Yaskawa INFORM job: A_ROOF_UPPER_0614_2_PAINT_65.JBI

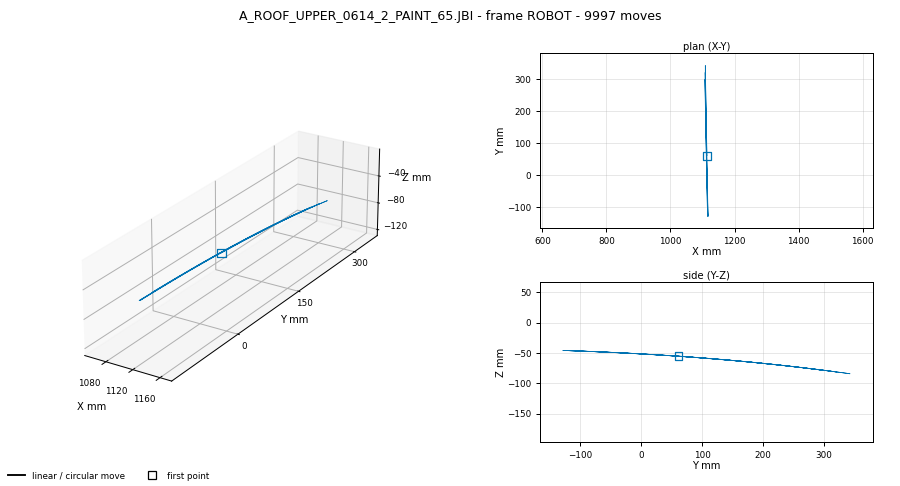
[picture p0: tool path of A_ROOF_UPPER_0614_2_PAINT_65.JBI in frame ROBOT, 9997 of 9997 moves have a stored position in this frame; points joined in program order, loops and branches not executed]
/JOB
//NAME A_ROOF_UPPER_0614_2_PAINT65
//POS
///NPOS 9997,0,0,0,0,0
///TOOL 1
///USER 0
///POSTYPE ROBOT
///RECTAN
///RCONF 1,0,0,0,0,0,0,0,0,0,0,0,0,0,0,0,0,0,0,0,0,0,0,0
C00000=1113.862,60.934,-55.122,179.977,7.455,149.407
C00001=1113.858,61.184,-55.139,179.979,7.459,149.407
C00002=1113.853,61.433,-55.156,179.980,7.462,149.408
C00003=1113.849,61.682,-55.174,179.981,7.466,149.408
C00004=1113.843,61.932,-55.191,179.983,7.470,149.409
C00005=1113.839,62.182,-55.208,179.984,7.475,149.409
C00006=1113.833,62.431,-55.225,179.985,7.478,149.410
C00007=1113.829,62.679,-55.242,179.986,7.483,149.410
C00008=1113.824,62.929,-55.259,179.988,7.487,149.411
C00009=1113.819,63.179,-55.276,179.989,7.491,149.411
C00010=1113.815,63.393,-55.291,179.990,7.494,149.412
C00011=1113.810,63.608,-55.306,179.991,7.497,149.412
C00012=1113.806,63.821,-55.321,179.992,7.500,149.413
C00013=1113.802,64.035,-55.336,179.993,7.504,149.413
C00014=1113.798,64.250,-55.351,179.994,7.507,149.414
C00015=1113.794,64.464,-55.366,179.995,7.510,149.414
C00016=1113.790,64.677,-55.380,179.997,7.514,149.415
C00017=1113.785,64.892,-55.395,179.998,7.518,149.415
C00018=1113.781,65.142,-55.412,179.999,7.521,149.415
C00019=1113.776,65.391,-55.429,-180.000,7.526,149.416
C00020=1113.771,65.641,-55.447,-179.998,7.530,149.417
C00021=1113.766,65.889,-55.464,-179.996,7.534,149.417
C00022=1113.761,66.138,-55.482,-179.995,7.538,149.418
C00023=1113.756,66.388,-55.499,-179.994,7.541,149.418
C00024=1113.751,66.637,-55.516,-179.993,7.545,149.418
C00025=1113.746,66.887,-55.533,-179.992,7.549,149.419
C00026=1113.741,67.136,-55.551,-179.990,7.553,149.420
C00027=1113.737,67.386,-55.568,-179.989,7.557,149.420
C00028=1113.732,67.635,-55.586,-179.987,7.561,149.421
C00029=1113.727,67.885,-55.603,-179.986,7.565,149.421
C00030=1113.722,68.134,-55.621,-179.985,7.569,149.422
C00031=1113.717,68.383,-55.638,-179.983,7.573,149.422
C00032=1113.712,68.632,-55.656,-179.982,7.576,149.423
C00033=1113.707,68.882,-55.673,-179.981,7.581,149.423
C00034=1113.702,69.131,-55.691,-179.980,7.585,149.424
C00035=1113.698,69.380,-55.709,-179.978,7.589,149.424
C00036=1113.693,69.630,-55.726,-179.976,7.592,149.425
C00037=1113.688,69.879,-55.744,-179.975,7.597,149.425
C00038=1113.682,70.128,-55.761,-179.974,7.601,149.426
C00039=1113.677,70.377,-55.779,-179.972,7.605,149.426
C00040=1113.673,70.626,-55.796,-179.971,7.609,149.427
C00041=1113.668,70.876,-55.813,-179.969,7.613,149.427
C00042=1113.663,71.125,-55.831,-179.969,7.616,149.428
C00043=1113.658,71.374,-55.849,-179.967,7.620,149.428
C00044=1113.653,71.625,-55.867,-179.966,7.624,149.429
C00045=1113.649,71.874,-55.884,-179.964,7.628,149.429
C00046=1113.644,72.123,-55.902,-179.963,7.632,149.430
C00047=1113.639,72.373,-55.920,-179.962,7.636,149.430
C00048=1113.634,72.622,-55.938,-179.960,7.640,149.431
C00049=1113.629,72.871,-55.956,-179.958,7.644,149.431
C00050=1113.624,73.120,-55.974,-179.957,7.648,149.432
C00051=1113.619,73.370,-55.991,-179.956,7.652,149.432
C00052=1113.614,73.619,-56.009,-179.954,7.656,149.433
C00053=1113.610,73.868,-56.026,-179.953,7.660,149.433
C00054=1113.605,74.117,-56.044,-179.952,7.663,149.434
C00055=1113.600,74.367,-56.062,-179.950,7.667,149.434
C00056=1113.595,74.616,-56.079,-179.949,7.671,149.434
C00057=1113.590,74.866,-56.097,-179.948,7.675,149.435
C00058=1113.585,75.115,-56.115,-179.946,7.679,149.436
C00059=1113.580,75.364,-56.133,-179.945,7.683,149.436
C00060=1113.575,75.613,-56.151,-179.944,7.688,149.437
C00061=1113.570,75.862,-56.169,-179.942,7.691,149.437
C00062=1113.566,76.113,-56.187,-179.940,7.695,149.437
C00063=1113.561,76.362,-56.205,-179.939,7.699,149.438
C00064=1113.556,76.611,-56.223,-179.938,7.704,149.439
C00065=1113.551,76.860,-56.241,-179.936,7.707,149.439
C00066=1113.547,77.074,-56.257,-179.935,7.711,149.439
C00067=1113.543,77.288,-56.272,-179.934,7.714,149.440
C00068=1113.539,77.503,-56.287,-179.934,7.717,149.441
C00069=1113.535,77.716,-56.303,-179.933,7.720,149.441
C00070=1113.531,77.931,-56.318,-179.932,7.723,149.441
C00071=1113.526,78.144,-56.334,-179.931,7.726,149.442
C00072=1113.522,78.359,-56.349,-179.930,7.729,149.442
C00073=1113.518,78.572,-56.365,-179.930,7.732,149.443
C00074=1113.513,78.822,-56.383,-179.928,7.736,149.443
C00075=1113.508,79.071,-56.401,-179.928,7.740,149.444
C00076=1113.504,79.321,-56.419,-179.926,7.744,149.444
C00077=1113.499,79.570,-56.437,-179.926,7.747,149.445
C00078=1113.494,79.819,-56.455,-179.924,7.751,149.445
C00079=1113.489,80.068,-56.473,-179.924,7.755,149.446
C00080=1113.484,80.317,-56.491,-179.922,7.758,149.447
C00081=1113.480,80.567,-56.509,-179.921,7.763,149.447
C00082=1113.475,80.816,-56.527,-179.920,7.766,149.448
C00083=1113.469,81.066,-56.546,-179.919,7.770,149.448
C00084=1113.464,81.315,-56.564,-179.918,7.773,149.449
C00085=1113.459,81.564,-56.582,-179.917,7.777,149.449
C00086=1113.455,81.814,-56.600,-179.916,7.781,149.450
C00087=1113.450,82.063,-56.618,-179.915,7.785,149.450
C00088=1113.445,82.312,-56.636,-179.914,7.788,149.451
C00089=1113.440,82.561,-56.655,-179.913,7.792,149.452
C00090=1113.436,82.810,-56.673,-179.911,7.796,149.452
C00091=1113.430,83.060,-56.692,-179.911,7.800,149.453
C00092=1113.426,83.310,-56.710,-179.909,7.804,149.453
C00093=1113.421,83.559,-56.728,-179.908,7.807,149.454
C00094=1113.416,83.808,-56.746,-179.907,7.811,149.454
C00095=1113.412,84.057,-56.765,-179.906,7.815,149.455
C00096=1113.407,84.306,-56.783,-179.905,7.818,149.455
C00097=1113.401,84.556,-56.801,-179.904,7.823,149.456
C00098=1113.396,84.805,-56.819,-179.902,7.827,149.456
C00099=1113.392,85.055,-56.838,-179.901,7.830,149.457
C00100=1113.387,85.303,-56.856,-179.900,7.834,149.457
C00101=1113.382,85.553,-56.874,-179.898,7.838,149.458
C00102=1113.377,85.802,-56.893,-179.898,7.841,149.458
C00103=1113.372,86.052,-56.911,-179.896,7.845,149.459
C00104=1113.368,86.301,-56.930,-179.895,7.849,149.459
C00105=1113.363,86.550,-56.948,-179.894,7.853,149.460
C00106=1113.357,86.799,-56.967,-179.893,7.856,149.460
C00107=1113.353,87.048,-56.986,-179.891,7.860,149.461
C00108=1113.348,87.298,-57.004,-179.890,7.864,149.461
C00109=1113.343,87.547,-57.022,-179.889,7.868,149.462
C00110=1113.339,87.796,-57.041,-179.887,7.872,149.462
C00111=1113.334,88.046,-57.059,-179.886,7.876,149.463
C00112=1113.329,88.295,-57.077,-179.885,7.879,149.463
C00113=1113.324,88.544,-57.097,-179.884,7.883,149.464
C00114=1113.319,88.793,-57.115,-179.882,7.887,149.464
C00115=1113.314,89.043,-57.133,-179.881,7.891,149.465
C00116=1113.310,89.292,-57.152,-179.880,7.894,149.465
C00117=1113.305,89.541,-57.170,-179.879,7.898,149.466
C00118=1113.300,89.790,-57.189,-179.877,7.902,149.466
C00119=1113.295,90.040,-57.208,-179.876,7.906,149.467
C00120=1113.290,90.289,-57.226,-179.875,7.909,149.467
C00121=1113.286,90.538,-57.245,-179.873,7.914,149.468
C00122=1113.282,90.752,-57.261,-179.872,7.916,149.468
C00123=1113.277,90.966,-57.277,-179.870,7.920,149.469
C00124=1113.273,91.180,-57.294,-179.869,7.923,149.469
C00125=1113.269,91.394,-57.309,-179.868,7.926,149.469
C00126=1113.265,91.609,-57.325,-179.867,7.930,149.470
C00127=1113.261,91.823,-57.341,-179.866,7.933,149.470
C00128=1113.257,92.036,-57.357,-179.865,7.937,149.471
C00129=1113.252,92.250,-57.373,-179.864,7.940,149.471
C00130=1113.248,92.500,-57.392,-179.862,7.944,149.472
C00131=1113.242,92.749,-57.411,-179.861,7.947,149.472
C00132=1113.238,92.998,-57.430,-179.859,7.951,149.472
C00133=1113.234,93.247,-57.449,-179.858,7.955,149.473
C00134=1113.228,93.497,-57.467,-179.856,7.959,149.473
C00135=1113.224,93.746,-57.486,-179.855,7.962,149.474
C00136=1113.218,93.995,-57.505,-179.854,7.967,149.474
C00137=1113.214,94.244,-57.524,-179.852,7.970,149.475
C00138=1113.209,94.493,-57.543,-179.851,7.974,149.475
C00139=1113.204,94.743,-57.561,-179.849,7.978,149.476
C00140=1113.199,94.992,-57.581,-179.847,7.982,149.476
C00141=1113.194,95.241,-57.599,-179.846,7.986,149.477
C00142=1113.190,95.491,-57.618,-179.844,7.990,149.477
C00143=1113.185,95.739,-57.637,-179.843,7.993,149.477
C00144=1113.180,95.989,-57.657,-179.842,7.997,149.478
C00145=1113.175,96.238,-57.675,-179.840,8.001,149.478
C00146=1113.171,96.488,-57.694,-179.838,8.005,149.479
C00147=1113.166,96.736,-57.713,-179.837,8.009,149.479
C00148=1113.160,96.986,-57.732,-179.835,8.012,149.480
C00149=1113.156,97.235,-57.751,-179.834,8.016,149.480
C00150=1113.151,97.484,-57.770,-179.832,8.020,149.481
C00151=1113.146,97.733,-57.790,-179.830,8.024,149.481
C00152=1113.141,97.983,-57.808,-179.829,8.028,149.481
C00153=1113.137,98.232,-57.827,-179.827,8.032,149.482
C00154=1113.132,98.481,-57.846,-179.825,8.035,149.482
C00155=1113.127,98.730,-57.866,-179.824,8.039,149.482
C00156=1113.123,98.980,-57.885,-179.822,8.043,149.483
C00157=1113.118,99.229,-57.903,-179.821,8.046,149.483
C00158=1113.113,99.479,-57.923,-179.819,8.050,149.484
C00159=1113.108,99.727,-57.942,-179.818,8.054,149.484
C00160=1113.104,99.977,-57.961,-179.816,8.058,149.485
C00161=1113.098,100.226,-57.981,-179.814,8.061,149.485
C00162=1113.094,100.475,-58.000,-179.813,8.065,149.485
C00163=1113.089,100.724,-58.019,-179.811,8.069,149.486
C00164=1113.084,100.973,-58.039,-179.809,8.073,149.486
C00165=1113.080,101.222,-58.057,-179.807,8.077,149.486
C00166=1113.075,101.471,-58.077,-179.806,8.080,149.487
C00167=1113.070,101.722,-58.096,-179.804,8.084,149.487
C00168=1113.065,101.970,-58.115,-179.802,8.088,149.488
C00169=1113.060,102.220,-58.134,-179.800,8.092,149.488
C00170=1113.055,102.469,-58.154,-179.799,8.096,149.488
C00171=1113.050,102.718,-58.173,-179.797,8.099,149.489
C00172=1113.046,102.967,-58.192,-179.795,8.103,149.489
C00173=1113.041,103.216,-58.212,-179.794,8.107,149.489
C00174=1113.036,103.466,-58.231,-179.792,8.111,149.490
C00175=1113.031,103.715,-58.251,-179.790,8.114,149.490
C00176=1113.027,103.963,-58.270,-179.788,8.119,149.491
C00177=1113.022,104.213,-58.290,-179.786,8.122,149.491
C00178=1113.018,104.427,-58.307,-179.785,8.126,149.491
C00179=1113.014,104.640,-58.323,-179.783,8.129,149.491
C00180=1113.009,104.855,-58.340,-179.781,8.132,149.492
C00181=1113.005,105.069,-58.356,-179.780,8.135,149.492
C00182=1113.001,105.282,-58.373,-179.778,8.138,149.492
C00183=1112.997,105.497,-58.389,-179.777,8.141,149.492
C00184=1112.993,105.710,-58.407,-179.775,8.145,149.493
C00185=1112.989,105.924,-58.423,-179.774,8.148,149.493
C00186=1112.985,106.173,-58.443,-179.771,8.152,149.493
C00187=1112.980,106.422,-58.463,-179.769,8.156,149.494
C00188=1112.975,106.672,-58.482,-179.767,8.159,149.494
C00189=1112.970,106.921,-58.502,-179.766,8.163,149.494
C00190=1112.965,107.171,-58.522,-179.764,8.167,149.495
C00191=1112.960,107.419,-58.542,-179.762,8.170,149.495
C00192=1112.956,107.668,-58.561,-179.760,8.174,149.495
C00193=1112.952,107.918,-58.580,-179.758,8.178,149.496
C00194=1112.946,108.167,-58.600,-179.756,8.181,149.496
C00195=1112.942,108.416,-58.620,-179.754,8.185,149.496
C00196=1112.937,108.665,-58.640,-179.752,8.189,149.496
C00197=1112.932,108.915,-58.659,-179.750,8.193,149.497
C00198=1112.927,109.163,-58.679,-179.748,8.197,149.497
C00199=1112.922,109.413,-58.699,-179.746,8.200,149.497
C00200=1112.918,109.662,-58.719,-179.744,8.204,149.498
C00201=1112.913,109.911,-58.739,-179.742,8.207,149.498
C00202=1112.908,110.160,-58.758,-179.740,8.211,149.498
C00203=1112.903,110.410,-58.778,-179.738,8.215,149.498
C00204=1112.899,110.659,-58.798,-179.736,8.218,149.499
C00205=1112.894,110.908,-58.818,-179.733,8.222,149.499
C00206=1112.889,111.157,-58.837,-179.731,8.226,149.499
C00207=1112.884,111.406,-58.858,-179.730,8.229,149.500
C00208=1112.879,111.656,-58.877,-179.728,8.232,149.500
C00209=1112.875,111.905,-58.898,-179.726,8.236,149.500
C00210=1112.870,112.153,-58.917,-179.725,8.240,149.500
C00211=1112.865,112.402,-58.937,-179.723,8.243,149.501
C00212=1112.861,112.652,-58.957,-179.721,8.246,149.501
C00213=1112.856,112.901,-58.977,-179.719,8.250,149.501
C00214=1112.851,113.150,-58.997,-179.717,8.253,149.502
C00215=1112.847,113.399,-59.017,-179.715,8.257,149.502
C00216=1112.842,113.648,-59.037,-179.714,8.260,149.502
C00217=1112.837,113.897,-59.057,-179.712,8.264,149.502
C00218=1112.832,114.147,-59.077,-179.710,8.267,149.503
C00219=1112.827,114.396,-59.098,-179.709,8.271,149.503
C00220=1112.822,114.646,-59.117,-179.707,8.274,149.503
C00221=1112.818,114.895,-59.138,-179.705,8.277,149.504
C00222=1112.813,115.143,-59.157,-179.703,8.281,149.504
C00223=1112.808,115.392,-59.177,-179.701,8.285,149.504
C00224=1112.804,115.641,-59.198,-179.700,8.287,149.504
C00225=1112.798,115.891,-59.218,-179.698,8.291,149.505
C00226=1112.794,116.140,-59.238,-179.696,8.295,149.505
C00227=1112.789,116.389,-59.259,-179.694,8.298,149.505
C00228=1112.785,116.639,-59.278,-179.693,8.301,149.506
C00229=1112.780,116.888,-59.299,-179.691,8.304,149.506
C00230=1112.775,117.136,-59.319,-179.689,8.308,149.506
C00231=1112.770,117.386,-59.339,-179.687,8.312,149.506
C00232=1112.765,117.635,-59.359,-179.686,8.314,149.507
C00233=1112.761,117.884,-59.380,-179.684,8.318,149.507
C00234=1112.757,118.097,-59.397,-179.683,8.321,149.507
C00235=1112.752,118.311,-59.415,-179.681,8.324,149.508
C00236=1112.749,118.526,-59.432,-179.679,8.327,149.508
C00237=1112.745,118.739,-59.449,-179.678,8.330,149.508
C00238=1112.741,118.953,-59.467,-179.676,8.333,149.508
C00239=1112.737,119.167,-59.484,-179.675,8.335,149.508
C00240=1112.732,119.381,-59.501,-179.673,8.338,149.509
C00241=1112.728,119.594,-59.519,-179.671,8.342,149.509
C00242=1112.724,119.843,-59.539,-179.670,8.344,149.509
C00243=1112.719,120.093,-59.560,-179.668,8.348,149.510
C00244=1112.714,120.342,-59.580,-179.666,8.352,149.510
C00245=1112.709,120.591,-59.600,-179.665,8.354,149.510
C00246=1112.705,120.840,-59.621,-179.663,8.358,149.510
C00247=1112.700,121.089,-59.641,-179.661,8.362,149.511
C00248=1112.695,121.338,-59.662,-179.659,8.365,149.511
C00249=1112.691,121.587,-59.682,-179.658,8.368,149.511
C00250=1112.686,121.836,-59.703,-179.655,8.372,149.511
C00251=1112.681,122.085,-59.724,-179.654,8.375,149.512
C00252=1112.677,122.335,-59.743,-179.652,8.378,149.512
C00253=1112.671,122.584,-59.764,-179.650,8.382,149.512
C00254=1112.667,122.833,-59.785,-179.648,8.385,149.513
C00255=1112.663,123.082,-59.805,-179.647,8.388,149.513
C00256=1112.657,123.331,-59.826,-179.645,8.392,149.513
C00257=1112.653,123.580,-59.846,-179.643,8.395,149.513
C00258=1112.648,123.830,-59.867,-179.641,8.399,149.514
C00259=1112.643,124.079,-59.888,-179.640,8.402,149.514
C00260=1112.639,124.328,-59.908,-179.638,8.405,149.514
C00261=1112.634,124.577,-59.929,-179.636,8.409,149.515
C00262=1112.629,124.826,-59.949,-179.635,8.412,149.515
C00263=1112.624,125.075,-59.970,-179.633,8.415,149.515
C00264=1112.620,125.324,-59.991,-179.631,8.419,149.515
C00265=1112.615,125.573,-60.011,-179.629,8.422,149.516
C00266=1112.611,125.823,-60.032,-179.627,8.425,149.516
C00267=1112.606,126.072,-60.053,-179.626,8.429,149.516
C00268=1112.601,126.320,-60.074,-179.624,8.432,149.517
C00269=1112.597,126.569,-60.095,-179.622,8.435,149.517
C00270=1112.592,126.819,-60.116,-179.620,8.439,149.517
C00271=1112.587,127.068,-60.136,-179.619,8.441,149.517
C00272=1112.582,127.317,-60.157,-179.617,8.445,149.518
C00273=1112.578,127.566,-60.177,-179.615,8.449,149.518
C00274=1112.572,127.815,-60.198,-179.614,8.451,149.518
C00275=1112.568,128.064,-60.219,-179.611,8.455,149.518
C00276=1112.563,128.313,-60.240,-179.610,8.459,149.519
C00277=1112.559,128.562,-60.261,-179.608,8.462,149.519
C00278=1112.554,128.812,-60.282,-179.606,8.465,149.519
C00279=1112.550,129.060,-60.303,-179.604,8.469,149.519
C00280=1112.545,129.310,-60.324,-179.603,8.472,149.520
C00281=1112.540,129.558,-60.345,-179.601,8.475,149.520
C00282=1112.535,129.807,-60.366,-179.599,8.479,149.520
C00283=1112.530,130.057,-60.387,-179.597,8.482,149.521
C00284=1112.526,130.306,-60.407,-179.596,8.485,149.521
C00285=1112.521,130.555,-60.429,-179.594,8.489,149.521
C00286=1112.517,130.804,-60.449,-179.592,8.492,149.521
C00287=1112.512,131.053,-60.470,-179.591,8.495,149.522
C00288=1112.507,131.302,-60.491,-179.589,8.499,149.522
C00289=1112.502,131.551,-60.512,-179.587,8.502,149.522
C00290=1112.498,131.765,-60.531,-179.585,8.505,149.523
C00291=1112.494,131.979,-60.549,-179.584,8.508,149.523
C00292=1112.490,132.192,-60.567,-179.582,8.510,149.523
C00293=1112.487,132.406,-60.585,-179.581,8.513,149.523
C00294=1112.483,132.619,-60.603,-179.580,8.516,149.524
C00295=1112.478,132.834,-60.621,-179.579,8.519,149.524
C00296=1112.474,133.047,-60.639,-179.576,8.522,149.524
C00297=1112.470,133.261,-60.658,-179.575,8.525,149.524
C00298=1112.465,133.510,-60.678,-179.574,8.528,149.525
C00299=1112.461,133.759,-60.699,-179.572,8.531,149.525
C00300=1112.456,134.008,-60.721,-179.570,8.535,149.525
C00301=1112.451,134.257,-60.742,-179.568,8.538,149.526
C00302=1112.446,134.506,-60.764,-179.566,8.541,149.526
C00303=1112.442,134.755,-60.784,-179.565,8.545,149.526
C00304=1112.438,135.004,-60.806,-179.563,8.548,149.526
C00305=1112.432,135.254,-60.827,-179.561,8.552,149.527
C00306=1112.428,135.502,-60.848,-179.560,8.555,149.527
C00307=1112.423,135.751,-60.869,-179.558,8.558,149.527
C00308=1112.419,136.001,-60.891,-179.556,8.562,149.528
C00309=1112.414,136.250,-60.912,-179.554,8.565,149.528
C00310=1112.410,136.498,-60.933,-179.553,8.568,149.528
C00311=1112.404,136.747,-60.954,-179.551,8.572,149.528
C00312=1112.400,136.997,-60.976,-179.549,8.576,149.529
C00313=1112.395,137.246,-60.997,-179.548,8.578,149.529
C00314=1112.390,137.495,-61.019,-179.546,8.582,149.529
C00315=1112.386,137.744,-61.039,-179.544,8.586,149.530
C00316=1112.381,137.993,-61.061,-179.543,8.588,149.530
C00317=1112.377,138.242,-61.083,-179.541,8.592,149.530
C00318=1112.371,138.491,-61.104,-179.539,8.596,149.531
C00319=1112.367,138.740,-61.126,-179.538,8.598,149.531
C00320=1112.363,138.988,-61.147,-179.535,8.602,149.531
C00321=1112.358,139.238,-61.168,-179.534,8.606,149.532
C00322=1112.354,139.487,-61.190,-179.532,8.609,149.532
C00323=1112.349,139.736,-61.212,-179.531,8.612,149.532
C00324=1112.343,139.985,-61.233,-179.529,8.616,149.532
C00325=1112.339,140.234,-61.255,-179.527,8.619,149.533
C00326=1112.334,140.483,-61.276,-179.526,8.622,149.533
C00327=1112.330,140.732,-61.297,-179.524,8.626,149.533
C00328=1112.326,140.981,-61.319,-179.523,8.629,149.534
C00329=1112.321,141.230,-61.340,-179.520,8.633,149.534
C00330=1112.317,141.479,-61.363,-179.519,8.636,149.535
C00331=1112.311,141.729,-61.383,-179.517,8.639,149.535
C00332=1112.306,141.977,-61.405,-179.515,8.643,149.535
C00333=1112.302,142.226,-61.427,-179.514,8.646,149.535
C00334=1112.297,142.475,-61.449,-179.512,8.649,149.536
C00335=1112.292,142.724,-61.470,-179.511,8.653,149.536
C00336=1112.288,142.974,-61.492,-179.508,8.657,149.536
C00337=1112.283,143.222,-61.514,-179.507,8.660,149.537
C00338=1112.279,143.472,-61.536,-179.505,8.663,149.537
C00339=1112.274,143.720,-61.557,-179.504,8.667,149.537
C00340=1112.269,143.969,-61.579,-179.502,8.670,149.538
C00341=1112.265,144.218,-61.601,-179.501,8.674,149.538
C00342=1112.260,144.468,-61.622,-179.499,8.677,149.538
C00343=1112.255,144.717,-61.644,-179.497,8.681,149.539
C00344=1112.250,144.966,-61.666,-179.495,8.684,149.539
C00345=1112.246,145.215,-61.688,-179.494,8.687,149.539
C00346=1112.242,145.428,-61.706,-179.492,8.690,149.540
C00347=1112.238,145.642,-61.725,-179.490,8.694,149.540
C00348=1112.235,145.855,-61.744,-179.488,8.697,149.540
C00349=1112.230,146.069,-61.763,-179.487,8.700,149.540
C00350=1112.226,146.282,-61.781,-179.485,8.703,149.541
C00351=1112.222,146.496,-61.800,-179.483,8.706,149.541
C00352=1112.218,146.709,-61.818,-179.481,8.710,149.541
C00353=1112.214,146.924,-61.837,-179.480,8.712,149.541
C00354=1112.209,147.172,-61.859,-179.478,8.716,149.542
C00355=1112.205,147.422,-61.881,-179.476,8.719,149.542
C00356=1112.200,147.670,-61.903,-179.474,8.723,149.542
C00357=1112.196,147.920,-61.925,-179.471,8.727,149.542
C00358=1112.190,148.169,-61.947,-179.469,8.731,149.542
C00359=1112.187,148.417,-61.970,-179.467,8.734,149.543
C00360=1112.182,148.666,-61.992,-179.465,8.737,149.543
C00361=1112.177,148.915,-62.014,-179.462,8.741,149.543
C00362=1112.173,149.164,-62.035,-179.460,8.744,149.543
C00363=1112.168,149.413,-62.057,-179.458,8.748,149.544
C00364=1112.163,149.662,-62.079,-179.456,8.751,149.544
C00365=1112.158,149.912,-62.102,-179.454,8.755,149.544
C00366=1112.154,150.160,-62.123,-179.452,8.758,149.544
C00367=1112.150,150.409,-62.146,-179.450,8.762,149.545
C00368=1112.145,150.658,-62.168,-179.448,8.765,149.545
C00369=1112.140,150.907,-62.190,-179.446,8.769,149.545
C00370=1112.135,151.156,-62.212,-179.444,8.772,149.545
C00371=1112.131,151.405,-62.234,-179.442,8.776,149.546
C00372=1112.127,151.654,-62.257,-179.440,8.779,149.546
C00373=1112.122,151.903,-62.279,-179.438,8.783,149.546
C00374=1112.117,152.152,-62.301,-179.435,8.786,149.546
C00375=1112.112,152.401,-62.323,-179.433,8.789,149.546
C00376=1112.108,152.650,-62.346,-179.431,8.793,149.547
C00377=1112.103,152.899,-62.368,-179.429,8.796,149.547
C00378=1112.098,153.148,-62.390,-179.427,8.800,149.547
C00379=1112.094,153.397,-62.413,-179.425,8.803,149.547
C00380=1112.089,153.645,-62.434,-179.422,8.806,149.547
C00381=1112.084,153.895,-62.457,-179.420,8.810,149.548
C00382=1112.080,154.144,-62.480,-179.418,8.813,149.548
C00383=1112.075,154.392,-62.502,-179.416,8.817,149.548
C00384=1112.070,154.642,-62.524,-179.414,8.820,149.548
C00385=1112.066,154.890,-62.547,-179.412,8.823,149.548
C00386=1112.061,155.139,-62.569,-179.410,8.826,149.549
C00387=1112.057,155.388,-62.592,-179.408,8.830,149.549
C00388=1112.052,155.637,-62.614,-179.405,8.833,149.549
C00389=1112.047,155.887,-62.636,-179.403,8.836,149.549
C00390=1112.043,156.135,-62.659,-179.401,8.840,149.549
C00391=1112.038,156.384,-62.681,-179.398,8.843,149.549
C00392=1112.033,156.633,-62.704,-179.396,8.846,149.550
C00393=1112.029,156.882,-62.726,-179.394,8.850,149.550
C00394=1112.024,157.131,-62.749,-179.392,8.852,149.550
C00395=1112.020,157.380,-62.771,-179.390,8.856,149.550
C00396=1112.016,157.629,-62.794,-179.388,8.859,149.550
C00397=1112.011,157.878,-62.817,-179.386,8.862,149.550
C00398=1112.006,158.126,-62.839,-179.384,8.866,149.551
C00399=1112.001,158.376,-62.862,-179.382,8.869,149.551
C00400=1111.997,158.625,-62.884,-179.379,8.872,149.551
C00401=1111.992,158.873,-62.907,-179.378,8.875,149.551
C00402=1111.988,159.087,-62.927,-179.375,8.878,149.551
C00403=1111.985,159.301,-62.946,-179.374,8.881,149.551
C00404=1111.981,159.514,-62.966,-179.372,8.883,149.551
C00405=1111.976,159.727,-62.985,-179.370,8.887,149.552
C00406=1111.972,159.941,-63.004,-179.368,8.889,149.552
C00407=1111.969,160.155,-63.024,-179.366,8.892,149.552
C00408=1111.965,160.368,-63.044,-179.364,8.894,149.552
C00409=1111.960,160.581,-63.063,-179.362,8.898,149.552
C00410=1111.956,160.830,-63.085,-179.360,8.901,149.552
C00411=1111.951,161.079,-63.108,-179.358,8.903,149.552
C00412=1111.947,161.328,-63.132,-179.356,8.907,149.552
C00413=1111.942,161.577,-63.154,-179.354,8.910,149.553
C00414=1111.937,161.826,-63.177,-179.351,8.913,149.553
C00415=1111.933,162.075,-63.200,-179.349,8.917,149.553
C00416=1111.929,162.324,-63.223,-179.347,8.919,149.553
C00417=1111.924,162.573,-63.245,-179.345,8.922,149.553
C00418=1111.919,162.822,-63.268,-179.343,8.926,149.553
C00419=1111.914,163.071,-63.291,-179.341,8.929,149.553
C00420=1111.910,163.319,-63.314,-179.338,8.932,149.554
C00421=1111.906,163.568,-63.338,-179.336,8.934,149.554
C00422=1111.901,163.818,-63.360,-179.334,8.938,149.554
C00423=1111.897,164.067,-63.383,-179.332,8.941,149.554
C00424=1111.891,164.315,-63.406,-179.329,8.945,149.554
C00425=1111.887,164.564,-63.429,-179.328,8.947,149.554
C00426=1111.883,164.813,-63.452,-179.325,8.950,149.554
C00427=1111.878,165.062,-63.475,-179.323,8.953,149.554
C00428=1111.874,165.311,-63.498,-179.320,8.957,149.554
C00429=1111.869,165.560,-63.522,-179.319,8.959,149.555
C00430=1111.864,165.808,-63.545,-179.316,8.962,149.555
C00431=1111.860,166.057,-63.567,-179.314,8.966,149.555
C00432=1111.855,166.306,-63.590,-179.312,8.969,149.555
C00433=1111.850,166.555,-63.613,-179.310,8.971,149.555
C00434=1111.846,166.804,-63.637,-179.308,8.975,149.555
C00435=1111.842,167.053,-63.659,-179.305,8.978,149.555
C00436=1111.837,167.302,-63.683,-179.303,8.981,149.555
C00437=1111.832,167.551,-63.706,-179.301,8.984,149.556
C00438=1111.828,167.800,-63.729,-179.299,8.987,149.556
C00439=1111.823,168.048,-63.752,-179.297,8.990,149.556
C00440=1111.818,168.297,-63.775,-179.295,8.993,149.556
C00441=1111.814,168.546,-63.799,-179.292,8.996,149.556
C00442=1111.809,168.795,-63.822,-179.290,8.999,149.556
C00443=1111.805,169.044,-63.846,-179.288,9.002,149.556
C00444=1111.801,169.292,-63.869,-179.286,9.005,149.556
C00445=1111.796,169.541,-63.892,-179.284,9.008,149.556
C00446=1111.791,169.791,-63.916,-179.281,9.011,149.556
C00447=1111.786,170.040,-63.939,-179.280,9.014,149.557
C00448=1111.782,170.289,-63.962,-179.277,9.017,149.557
C00449=1111.778,170.537,-63.985,-179.275,9.020,149.557
C00450=1111.773,170.786,-64.008,-179.273,9.023,149.557
C00451=1111.769,171.035,-64.032,-179.271,9.026,149.557
C00452=1111.764,171.284,-64.056,-179.268,9.029,149.557
C00453=1111.759,171.533,-64.079,-179.266,9.033,149.557
C00454=1111.755,171.782,-64.103,-179.264,9.035,149.557
C00455=1111.750,172.031,-64.126,-179.262,9.038,149.557
C00456=1111.746,172.279,-64.150,-179.260,9.042,149.558
C00457=1111.741,172.528,-64.173,-179.258,9.044,149.558
C00458=1111.737,172.742,-64.193,-179.256,9.046,149.558
C00459=1111.733,172.955,-64.213,-179.253,9.049,149.558
C00460=1111.729,173.168,-64.233,-179.252,9.052,149.558
C00461=1111.725,173.382,-64.253,-179.250,9.054,149.558
C00462=1111.721,173.595,-64.273,-179.248,9.057,149.558
C00463=1111.717,173.808,-64.294,-179.247,9.059,149.558
C00464=1111.714,174.022,-64.314,-179.245,9.062,149.558
C00465=1111.709,174.235,-64.334,-179.243,9.064,149.558
C00466=1111.705,174.484,-64.358,-179.240,9.067,149.558
C00467=1111.700,174.733,-64.381,-179.238,9.071,149.559
C00468=1111.695,174.982,-64.405,-179.236,9.073,149.559
C00469=1111.691,175.230,-64.429,-179.234,9.076,149.559
C00470=1111.686,175.479,-64.452,-179.232,9.080,149.559
C00471=1111.682,175.728,-64.476,-179.230,9.082,149.559
C00472=1111.677,175.977,-64.500,-179.227,9.085,149.559
C00473=1111.673,176.227,-64.523,-179.225,9.089,149.559
C00474=1111.669,176.475,-64.547,-179.223,9.091,149.559
C00475=1111.664,176.724,-64.571,-179.221,9.094,149.559
C00476=1111.660,176.972,-64.595,-179.219,9.097,149.560
C00477=1111.655,177.221,-64.618,-179.217,9.100,149.560
C00478=1111.651,177.470,-64.642,-179.214,9.103,149.560
C00479=1111.646,177.719,-64.666,-179.212,9.106,149.560
C00480=1111.641,177.967,-64.690,-179.210,9.109,149.560
C00481=1111.637,178.216,-64.713,-179.208,9.112,149.560
C00482=1111.632,178.465,-64.737,-179.206,9.115,149.560
C00483=1111.628,178.714,-64.761,-179.204,9.118,149.560
C00484=1111.624,178.963,-64.785,-179.201,9.121,149.560
C00485=1111.619,179.212,-64.808,-179.200,9.123,149.561
C00486=1111.615,179.460,-64.832,-179.197,9.127,149.561
C00487=1111.609,179.710,-64.856,-179.195,9.130,149.561
C00488=1111.605,179.958,-64.880,-179.192,9.133,149.561
C00489=1111.601,180.207,-64.905,-179.190,9.136,149.561
C00490=1111.596,180.456,-64.928,-179.187,9.139,149.561
C00491=1111.592,180.705,-64.952,-179.185,9.142,149.561
C00492=1111.588,180.953,-64.976,-179.182,9.145,149.561
C00493=1111.583,181.202,-65.000,-179.180,9.148,149.561
C00494=1111.578,181.451,-65.024,-179.178,9.151,149.561
C00495=1111.574,181.700,-65.049,-179.176,9.154,149.561
C00496=1111.569,181.949,-65.072,-179.173,9.157,149.561
C00497=1111.565,182.197,-65.096,-179.171,9.160,149.561
C00498=1111.561,182.446,-65.120,-179.168,9.163,149.561
C00499=1111.555,182.695,-65.144,-179.166,9.167,149.561
C00500=1111.551,182.944,-65.169,-179.164,9.169,149.561
C00501=1111.547,183.193,-65.193,-179.161,9.172,149.561
C00502=1111.542,183.441,-65.217,-179.159,9.175,149.562
C00503=1111.537,183.690,-65.241,-179.156,9.178,149.562
C00504=1111.533,183.939,-65.265,-179.154,9.181,149.562
C00505=1111.529,184.188,-65.289,-179.152,9.184,149.562
C00506=1111.524,184.436,-65.313,-179.149,9.187,149.562
C00507=1111.519,184.685,-65.338,-179.147,9.190,149.562
C00508=1111.515,184.934,-65.361,-179.144,9.192,149.562
C00509=1111.511,185.183,-65.386,-179.142,9.195,149.562
C00510=1111.506,185.432,-65.411,-179.139,9.198,149.562
C00511=1111.501,185.680,-65.435,-179.137,9.200,149.562
C00512=1111.497,185.929,-65.459,-179.135,9.204,149.562
C00513=1111.492,186.178,-65.484,-179.132,9.207,149.562
C00514=1111.489,186.391,-65.504,-179.130,9.209,149.562
C00515=1111.485,186.604,-65.525,-179.129,9.211,149.562
C00516=1111.481,186.818,-65.547,-179.127,9.214,149.562
C00517=1111.477,187.031,-65.566,-179.125,9.216,149.562
C00518=1111.473,187.244,-65.587,-179.122,9.219,149.562
C00519=1111.470,187.458,-65.608,-179.120,9.221,149.562
C00520=1111.465,187.671,-65.629,-179.118,9.224,149.562
C00521=1111.461,187.885,-65.651,-179.117,9.226,149.562
C00522=1111.457,188.133,-65.675,-179.114,9.229,149.562
C00523=1111.452,188.382,-65.700,-179.112,9.232,149.562
C00524=1111.448,188.631,-65.724,-179.110,9.235,149.562
C00525=1111.444,188.879,-65.748,-179.108,9.237,149.562
C00526=1111.438,189.128,-65.772,-179.105,9.240,149.562
C00527=1111.435,189.377,-65.797,-179.103,9.243,149.562
C00528=1111.429,189.626,-65.822,-179.101,9.245,149.562
C00529=1111.425,189.874,-65.846,-179.098,9.249,149.562
C00530=1111.421,190.123,-65.871,-179.096,9.251,149.562
C00531=1111.416,190.371,-65.895,-179.094,9.254,149.563
C00532=1111.412,190.621,-65.921,-179.091,9.257,149.563
C00533=1111.408,190.869,-65.945,-179.089,9.259,149.563
C00534=1111.402,191.118,-65.969,-179.087,9.263,149.563
C00535=1111.399,191.367,-65.994,-179.085,9.265,149.563
C00536=1111.393,191.616,-66.018,-179.083,9.268,149.563
C00537=1111.389,191.864,-66.042,-179.081,9.270,149.563
C00538=1111.385,192.113,-66.068,-179.078,9.273,149.563
C00539=1111.380,192.361,-66.092,-179.077,9.276,149.563
C00540=1111.376,192.611,-66.117,-179.074,9.279,149.563
C00541=1111.372,192.859,-66.141,-179.072,9.282,149.563
C00542=1111.366,193.108,-66.166,-179.070,9.285,149.563
C00543=1111.362,193.357,-66.192,-179.067,9.288,149.563
C00544=1111.358,193.605,-66.216,-179.065,9.290,149.563
C00545=1111.353,193.855,-66.241,-179.063,9.293,149.563
C00546=1111.349,194.103,-66.265,-179.061,9.296,149.564
C00547=1111.345,194.352,-66.291,-179.059,9.299,149.564
C00548=1111.340,194.601,-66.315,-179.057,9.301,149.564
C00549=1111.335,194.849,-66.339,-179.054,9.305,149.564
C00550=1111.331,195.098,-66.365,-179.053,9.307,149.564
C00551=1111.327,195.346,-66.389,-179.050,9.310,149.564
C00552=1111.322,195.596,-66.414,-179.048,9.313,149.564
C00553=1111.317,195.844,-66.440,-179.046,9.316,149.564
C00554=1111.313,196.093,-66.464,-179.044,9.318,149.564
C00555=1111.308,196.342,-66.489,-179.042,9.322,149.564
C00556=1111.304,196.590,-66.515,-179.039,9.325,149.564
C00557=1111.300,196.839,-66.539,-179.037,9.328,149.565
C00558=1111.295,197.088,-66.564,-179.034,9.331,149.565
C00559=1111.290,197.336,-66.589,-179.032,9.334,149.565
C00560=1111.286,197.585,-66.614,-179.029,9.337,149.565
C00561=1111.282,197.834,-66.639,-179.026,9.340,149.565
C00562=1111.277,198.083,-66.664,-179.024,9.343,149.565
C00563=1111.273,198.331,-66.689,-179.021,9.346,149.565
C00564=1111.268,198.580,-66.714,-179.019,9.349,149.565
C00565=1111.264,198.828,-66.739,-179.016,9.352,149.565
C00566=1111.259,199.078,-66.764,-179.013,9.355,149.565
C00567=1111.255,199.326,-66.789,-179.011,9.358,149.565
C00568=1111.250,199.575,-66.814,-179.008,9.361,149.565
C00569=1111.246,199.823,-66.839,-179.005,9.364,149.565
C00570=1111.242,200.037,-66.861,-179.002,9.367,149.564
C00571=1111.238,200.250,-66.883,-179.000,9.369,149.564
C00572=1111.234,200.463,-66.904,-178.999,9.371,149.565
C00573=1111.231,200.676,-66.926,-178.996,9.374,149.564
C00574=1111.226,200.889,-66.947,-178.994,9.377,149.564
C00575=1111.223,201.103,-66.969,-178.991,9.379,149.564
C00576=1111.219,201.315,-66.991,-178.989,9.382,149.564
C00577=1111.215,201.529,-67.012,-178.986,9.384,149.564
C00578=1111.211,201.777,-67.038,-178.983,9.387,149.564
C00579=1111.207,202.027,-67.062,-178.980,9.390,149.564
C00580=1111.202,202.275,-67.088,-178.978,9.393,149.564
C00581=1111.198,202.523,-67.114,-178.975,9.396,149.564
C00582=1111.193,202.772,-67.139,-178.972,9.399,149.564
C00583=1111.189,203.021,-67.164,-178.969,9.402,149.564
C00584=1111.184,203.270,-67.190,-178.967,9.405,149.564
C00585=1111.180,203.518,-67.215,-178.964,9.407,149.564
C00586=1111.175,203.767,-67.241,-178.961,9.410,149.563
C00587=1111.171,204.016,-67.266,-178.958,9.413,149.564
C00588=1111.167,204.264,-67.291,-178.955,9.416,149.563
C00589=1111.162,204.513,-67.316,-178.952,9.419,149.563
C00590=1111.158,204.761,-67.342,-178.949,9.421,149.563
C00591=1111.153,205.010,-67.368,-178.947,9.425,149.563
C00592=1111.149,205.259,-67.393,-178.944,9.427,149.563
C00593=1111.144,205.507,-67.418,-178.941,9.430,149.563
C00594=1111.140,205.756,-67.444,-178.938,9.433,149.563
C00595=1111.136,206.005,-67.470,-178.935,9.436,149.563
C00596=1111.131,206.254,-67.495,-178.932,9.439,149.563
C00597=1111.127,206.502,-67.521,-178.929,9.442,149.563
C00598=1111.122,206.750,-67.546,-178.926,9.445,149.562
C00599=1111.118,206.999,-67.572,-178.923,9.448,149.562
C00600=1111.113,207.248,-67.598,-178.920,9.451,149.562
C00601=1111.108,207.497,-67.624,-178.918,9.454,149.562
C00602=1111.104,207.745,-67.650,-178.915,9.456,149.562
C00603=1111.099,207.993,-67.675,-178.912,9.459,149.562
C00604=1111.095,208.242,-67.701,-178.909,9.462,149.562
C00605=1111.091,208.491,-67.727,-178.906,9.465,149.562
C00606=1111.087,208.740,-67.752,-178.903,9.469,149.562
C00607=1111.082,208.988,-67.778,-178.900,9.471,149.562
C00608=1111.078,209.237,-67.803,-178.897,9.474,149.562
C00609=1111.073,209.486,-67.829,-178.895,9.477,149.562
C00610=1111.069,209.734,-67.855,-178.892,9.480,149.561
C00611=1111.064,209.983,-67.881,-178.888,9.484,149.561
C00612=1111.059,210.232,-67.907,-178.886,9.487,149.561
C00613=1111.055,210.480,-67.933,-178.883,9.489,149.561
C00614=1111.051,210.729,-67.959,-178.880,9.492,149.561
C00615=1111.047,210.977,-67.985,-178.877,9.495,149.561
C00616=1111.043,211.226,-68.010,-178.874,9.499,149.561
C00617=1111.037,211.475,-68.036,-178.871,9.502,149.561
C00618=1111.033,211.723,-68.063,-178.868,9.505,149.561
C00619=1111.029,211.972,-68.089,-178.865,9.509,149.561
C00620=1111.025,212.220,-68.114,-178.862,9.511,149.561
C00621=1111.020,212.470,-68.141,-178.859,9.514,149.561
C00622=1111.016,212.718,-68.167,-178.856,9.518,149.561
C00623=1111.011,212.966,-68.193,-178.853,9.521,149.561
C00624=1111.007,213.215,-68.218,-178.851,9.524,149.561
C00625=1111.002,213.464,-68.245,-178.847,9.528,149.561
C00626=1110.999,213.676,-68.268,-178.846,9.530,149.561
C00627=1110.995,213.889,-68.289,-178.844,9.533,149.561
C00628=1110.991,214.103,-68.312,-178.842,9.535,149.561
C00629=1110.987,214.315,-68.334,-178.840,9.537,149.561
C00630=1110.984,214.529,-68.356,-178.838,9.540,149.561
C00631=1110.980,214.742,-68.380,-178.837,9.542,149.562
C00632=1110.976,214.954,-68.401,-178.834,9.546,149.562
C00633=1110.972,215.168,-68.424,-178.832,9.548,149.562
C00634=1110.968,215.417,-68.450,-178.830,9.550,149.562
C00635=1110.964,215.665,-68.476,-178.828,9.553,149.562
C00636=1110.959,215.914,-68.503,-178.826,9.557,149.562
C00637=1110.955,216.162,-68.529,-178.823,9.560,149.562
C00638=1110.951,216.411,-68.555,-178.821,9.562,149.562
C00639=1110.946,216.659,-68.582,-178.819,9.565,149.562
C00640=1110.941,216.908,-68.607,-178.817,9.569,149.563
C00641=1110.937,217.156,-68.634,-178.814,9.572,149.563
C00642=1110.932,217.405,-68.660,-178.812,9.574,149.563
C00643=1110.929,217.653,-68.687,-178.810,9.577,149.563
C00644=1110.924,217.902,-68.713,-178.808,9.581,149.563
C00645=1110.920,218.150,-68.740,-178.805,9.584,149.563
C00646=1110.915,218.400,-68.766,-178.803,9.586,149.563
C00647=1110.911,218.648,-68.792,-178.801,9.589,149.563
C00648=1110.907,218.896,-68.819,-178.798,9.593,149.563
C00649=1110.902,219.145,-68.845,-178.796,9.596,149.563
C00650=1110.898,219.393,-68.872,-178.794,9.599,149.564
C00651=1110.893,219.642,-68.898,-178.791,9.602,149.564
C00652=1110.889,219.890,-68.924,-178.789,9.605,149.564
C00653=1110.884,220.139,-68.952,-178.787,9.608,149.564
C00654=1110.880,220.388,-68.977,-178.785,9.611,149.564
C00655=1110.876,220.636,-69.004,-178.782,9.614,149.564
C00656=1110.872,220.884,-69.031,-178.779,9.617,149.564
C00657=1110.867,221.134,-69.057,-178.777,9.620,149.564
C00658=1110.863,221.382,-69.084,-178.774,9.624,149.564
C00659=1110.858,221.630,-69.111,-178.772,9.627,149.564
C00660=1110.854,221.878,-69.137,-178.770,9.629,149.564
C00661=1110.849,222.128,-69.164,-178.768,9.633,149.565
C00662=1110.845,222.376,-69.190,-178.765,9.636,149.565
C00663=1110.841,222.624,-69.217,-178.763,9.639,149.565
C00664=1110.836,222.873,-69.244,-178.760,9.642,149.565
C00665=1110.832,223.122,-69.270,-178.758,9.645,149.565
C00666=1110.827,223.370,-69.297,-178.755,9.648,149.565
C00667=1110.824,223.619,-69.324,-178.753,9.651,149.565
C00668=1110.819,223.867,-69.351,-178.750,9.654,149.565
C00669=1110.815,224.116,-69.378,-178.748,9.657,149.565
C00670=1110.811,224.364,-69.404,-178.745,9.661,149.565
C00671=1110.806,224.613,-69.431,-178.743,9.664,149.565
C00672=1110.801,224.862,-69.458,-178.740,9.667,149.565
C00673=1110.797,225.110,-69.484,-178.738,9.670,149.565
C00674=1110.792,225.358,-69.511,-178.735,9.673,149.566
C00675=1110.788,225.607,-69.538,-178.732,9.676,149.565
C00676=1110.784,225.855,-69.565,-178.730,9.679,149.565
C00677=1110.780,226.104,-69.592,-178.728,9.681,149.566
C00678=1110.775,226.353,-69.619,-178.725,9.684,149.566
C00679=1110.771,226.601,-69.646,-178.723,9.687,149.566
C00680=1110.767,226.849,-69.673,-178.720,9.690,149.566
C00681=1110.762,227.098,-69.700,-178.717,9.693,149.566
C00682=1110.759,227.311,-69.723,-178.715,9.696,149.566
C00683=1110.755,227.524,-69.746,-178.713,9.699,149.566
C00684=1110.751,227.737,-69.769,-178.710,9.702,149.566
C00685=1110.747,227.950,-69.792,-178.708,9.704,149.566
C00686=1110.744,228.162,-69.815,-178.706,9.706,149.566
C00687=1110.740,228.375,-69.839,-178.704,9.709,149.566
C00688=1110.736,228.588,-69.862,-178.701,9.711,149.566
C00689=1110.732,228.802,-69.885,-178.699,9.714,149.566
C00690=1110.728,229.050,-69.913,-178.696,9.717,149.566
C00691=1110.724,229.298,-69.939,-178.693,9.720,149.566
C00692=1110.719,229.547,-69.966,-178.691,9.723,149.566
C00693=1110.715,229.795,-69.993,-178.688,9.726,149.566
C00694=1110.710,230.044,-70.020,-178.685,9.729,149.565
C00695=1110.706,230.293,-70.048,-178.682,9.732,149.566
C00696=1110.701,230.541,-70.075,-178.679,9.735,149.565
C00697=1110.698,230.789,-70.102,-178.677,9.738,149.565
C00698=1110.693,231.037,-70.129,-178.674,9.740,149.565
C00699=1110.689,231.287,-70.157,-178.672,9.742,149.565
C00700=1110.684,231.535,-70.184,-178.669,9.746,149.565
C00701=1110.680,231.783,-70.211,-178.666,9.748,149.565
C00702=1110.675,232.031,-70.238,-178.663,9.751,149.565
C00703=1110.671,232.281,-70.266,-178.661,9.754,149.565
C00704=1110.667,232.529,-70.293,-178.658,9.757,149.565
C00705=1110.663,232.777,-70.320,-178.655,9.760,149.565
C00706=1110.658,233.025,-70.347,-178.652,9.763,149.565
C00707=1110.654,233.274,-70.375,-178.650,9.765,149.565
C00708=1110.650,233.522,-70.402,-178.647,9.767,149.565
C00709=1110.645,233.771,-70.429,-178.644,9.770,149.565
C00710=1110.642,234.019,-70.458,-178.641,9.773,149.565
C00711=1110.637,234.268,-70.485,-178.638,9.776,149.565
C00712=1110.632,234.516,-70.512,-178.636,9.778,149.564
C00713=1110.628,234.764,-70.539,-178.633,9.781,149.564
C00714=1110.624,235.013,-70.567,-178.631,9.784,149.564
C00715=1110.619,235.261,-70.595,-178.628,9.787,149.564
C00716=1110.615,235.510,-70.622,-178.625,9.789,149.564
C00717=1110.611,235.758,-70.650,-178.622,9.791,149.564
C00718=1110.606,236.007,-70.677,-178.620,9.794,149.564
C00719=1110.602,236.255,-70.705,-178.617,9.797,149.564
C00720=1110.598,236.504,-70.732,-178.615,9.799,149.564
C00721=1110.594,236.752,-70.760,-178.612,9.802,149.564
C00722=1110.590,237.001,-70.787,-178.609,9.805,149.563
C00723=1110.585,237.249,-70.815,-178.606,9.807,149.563
C00724=1110.581,237.497,-70.842,-178.604,9.810,149.563
C00725=1110.576,237.746,-70.871,-178.601,9.813,149.563
C00726=1110.571,237.995,-70.898,-178.598,9.815,149.563
C00727=1110.567,238.243,-70.926,-178.596,9.817,149.563
C00728=1110.563,238.491,-70.954,-178.593,9.820,149.563
C00729=1110.559,238.740,-70.981,-178.590,9.823,149.563
C00730=1110.555,238.988,-71.009,-178.588,9.825,149.563
C00731=1110.551,239.236,-71.037,-178.585,9.828,149.563
C00732=1110.546,239.485,-71.064,-178.583,9.831,149.563
C00733=1110.541,239.733,-71.093,-178.580,9.833,149.563
C00734=1110.537,239.981,-71.120,-178.577,9.836,149.563
C00735=1110.533,240.231,-71.148,-178.575,9.838,149.562
C00736=1110.529,240.478,-71.176,-178.572,9.841,149.563
C00737=1110.524,240.726,-71.203,-178.569,9.844,149.562
C00738=1110.521,240.939,-71.227,-178.567,9.846,149.562
C00739=1110.517,241.152,-71.250,-178.565,9.848,149.562
C00740=1110.513,241.365,-71.275,-178.563,9.850,149.562
C00741=1110.509,241.578,-71.299,-178.561,9.852,149.562
C00742=1110.506,241.791,-71.323,-178.559,9.854,149.562
C00743=1110.502,242.004,-71.347,-178.557,9.856,149.562
C00744=1110.499,242.217,-71.371,-178.555,9.858,149.562
C00745=1110.495,242.430,-71.395,-178.552,9.862,149.562
C00746=1110.490,242.678,-71.423,-178.550,9.864,149.562
C00747=1110.486,242.926,-71.451,-178.547,9.866,149.562
C00748=1110.482,243.174,-71.479,-178.545,9.869,149.562
C00749=1110.478,243.423,-71.507,-178.542,9.871,149.562
C00750=1110.473,243.672,-71.535,-178.539,9.874,149.562
C00751=1110.469,243.920,-71.563,-178.537,9.876,149.562
C00752=1110.465,244.168,-71.591,-178.535,9.880,149.562
C00753=1110.461,244.417,-71.619,-178.533,9.882,149.562
C00754=1110.456,244.665,-71.647,-178.530,9.885,149.562
C00755=1110.452,244.913,-71.675,-178.527,9.888,149.562
C00756=1110.448,245.161,-71.703,-178.525,9.890,149.562
C00757=1110.443,245.410,-71.732,-178.522,9.893,149.562
C00758=1110.439,245.658,-71.760,-178.520,9.895,149.562
C00759=1110.435,245.907,-71.788,-178.518,9.898,149.562
C00760=1110.430,246.155,-71.816,-178.515,9.901,149.562
C00761=1110.426,246.403,-71.844,-178.513,9.903,149.562
C00762=1110.421,246.652,-71.873,-178.511,9.906,149.562
C00763=1110.418,246.900,-71.901,-178.509,9.909,149.562
C00764=1110.413,247.148,-71.928,-178.506,9.912,149.562
C00765=1110.409,247.397,-71.957,-178.503,9.915,149.562
C00766=1110.404,247.645,-71.985,-178.501,9.918,149.562
C00767=1110.400,247.894,-72.014,-178.498,9.921,149.562
C00768=1110.396,248.142,-72.042,-178.494,9.924,149.562
C00769=1110.392,248.390,-72.070,-178.491,9.928,149.562
C00770=1110.387,248.639,-72.098,-178.488,9.930,149.562
C00771=1110.383,248.887,-72.126,-178.484,9.934,149.562
C00772=1110.379,249.135,-72.156,-178.481,9.937,149.561
C00773=1110.375,249.384,-72.184,-178.478,9.939,149.561
C00774=1110.370,249.632,-72.212,-178.474,9.943,149.561
C00775=1110.366,249.880,-72.240,-178.471,9.945,149.561
C00776=1110.361,250.129,-72.269,-178.468,9.948,149.561
C00777=1110.358,250.377,-72.298,-178.465,9.951,149.561
C00778=1110.353,250.626,-72.326,-178.462,9.953,149.560
C00779=1110.349,250.873,-72.354,-178.459,9.956,149.560
C00780=1110.344,251.122,-72.383,-178.456,9.959,149.560
C00781=1110.341,251.370,-72.412,-178.453,9.961,149.560
C00782=1110.336,251.618,-72.440,-178.450,9.963,149.560
C00783=1110.332,251.867,-72.468,-178.448,9.966,149.560
C00784=1110.328,252.115,-72.498,-178.444,9.968,149.559
C00785=1110.323,252.363,-72.526,-178.441,9.971,149.559
C00786=1110.319,252.612,-72.554,-178.439,9.973,149.559
C00787=1110.315,252.860,-72.584,-178.436,9.976,149.559
C00788=1110.311,253.108,-72.611,-178.434,9.978,149.559
C00789=1110.306,253.357,-72.640,-178.431,9.981,149.559
C00790=1110.302,253.605,-72.670,-178.428,9.982,149.559
C00791=1110.298,253.854,-72.698,-178.425,9.985,149.558
C00792=1110.293,254.101,-72.727,-178.423,9.987,149.558
C00793=1110.290,254.350,-72.755,-178.420,9.990,149.558
C00794=1110.285,254.563,-72.780,-178.418,9.992,149.558
C00795=1110.282,254.775,-72.804,-178.416,9.993,149.558
C00796=1110.278,254.989,-72.829,-178.414,9.995,149.558
C00797=1110.274,255.201,-72.854,-178.412,9.997,149.558
C00798=1110.271,255.414,-72.878,-178.410,10.000,149.558
C00799=1110.267,255.626,-72.903,-178.408,10.002,149.558
C00800=1110.264,255.839,-72.928,-178.407,10.003,149.558
C00801=1110.260,256.052,-72.953,-178.405,10.006,149.558
C00802=1110.256,256.300,-72.981,-178.402,10.008,149.558
C00803=1110.251,256.548,-73.010,-178.399,10.011,149.558
C00804=1110.247,256.797,-73.039,-178.396,10.014,149.558
C00805=1110.244,257.045,-73.068,-178.393,10.017,149.558
C00806=1110.239,257.293,-73.097,-178.390,10.020,149.558
C00807=1110.234,257.541,-73.126,-178.389,10.022,149.558
C00808=1110.230,257.789,-73.155,-178.386,10.025,149.558
C00809=1110.226,258.038,-73.183,-178.383,10.028,149.557
C00810=1110.222,258.286,-73.213,-178.380,10.030,149.557
C00811=1110.218,258.535,-73.242,-178.377,10.034,149.557
C00812=1110.213,258.783,-73.271,-178.374,10.036,149.557
C00813=1110.209,259.031,-73.300,-178.371,10.039,149.557
C00814=1110.205,259.279,-73.329,-178.368,10.042,149.557
C00815=1110.201,259.528,-73.358,-178.365,10.045,149.557
C00816=1110.197,259.776,-73.387,-178.363,10.047,149.557
C00817=1110.192,260.023,-73.416,-178.361,10.050,149.557
C00818=1110.187,260.272,-73.445,-178.358,10.052,149.557
C00819=1110.184,260.520,-73.474,-178.355,10.055,149.557
C00820=1110.180,260.769,-73.503,-178.352,10.058,149.557
C00821=1110.176,261.017,-73.533,-178.349,10.061,149.557
C00822=1110.171,261.266,-73.561,-178.346,10.063,149.556
C00823=1110.167,261.514,-73.591,-178.343,10.066,149.556
C00824=1110.162,261.762,-73.620,-178.340,10.069,149.556
C00825=1110.158,262.010,-73.649,-178.337,10.072,149.556
C00826=1110.154,262.258,-73.679,-178.334,10.074,149.556
C00827=1110.150,262.506,-73.708,-178.331,10.077,149.556
C00828=1110.145,262.755,-73.738,-178.328,10.080,149.556
C00829=1110.142,263.003,-73.766,-178.326,10.082,149.556
C00830=1110.137,263.252,-73.795,-178.323,10.085,149.556
C00831=1110.133,263.500,-73.825,-178.320,10.087,149.555
C00832=1110.129,263.748,-73.854,-178.317,10.090,149.555
C00833=1110.124,263.996,-73.883,-178.314,10.093,149.555
C00834=1110.120,264.244,-73.913,-178.311,10.095,149.555
C00835=1110.116,264.492,-73.942,-178.308,10.098,149.555
C00836=1110.112,264.740,-73.972,-178.305,10.101,149.555
C00837=1110.108,264.989,-74.001,-178.303,10.103,149.555
C00838=1110.103,265.237,-74.031,-178.299,10.105,149.554
C00839=1110.099,265.485,-74.060,-178.296,10.108,149.554
C00840=1110.095,265.733,-74.090,-178.293,10.111,149.554
C00841=1110.091,265.982,-74.119,-178.291,10.113,149.554
C00842=1110.086,266.230,-74.149,-178.288,10.116,149.554
C00843=1110.082,266.479,-74.179,-178.285,10.118,149.554
C00844=1110.078,266.727,-74.208,-178.282,10.121,149.554
C00845=1110.073,266.975,-74.237,-178.280,10.123,149.554
C00846=1110.069,267.223,-74.268,-178.277,10.126,149.553
C00847=1110.065,267.471,-74.297,-178.274,10.129,149.553
C00848=1110.061,267.719,-74.326,-178.271,10.131,149.553
C00849=1110.057,267.968,-74.356,-178.269,10.133,149.553
C00850=1110.053,268.180,-74.381,-178.266,10.136,149.553
C00851=1110.050,268.393,-74.407,-178.264,10.138,149.553
C00852=1110.046,268.605,-74.432,-178.261,10.140,149.553
C00853=1110.042,268.817,-74.458,-178.259,10.142,149.553
C00854=1110.038,269.031,-74.483,-178.256,10.145,149.553
C00855=1110.035,269.242,-74.508,-178.254,10.147,149.552
C00856=1110.032,269.455,-74.534,-178.251,10.149,149.552
C00857=1110.028,269.667,-74.559,-178.250,10.151,149.552
C00858=1110.024,269.916,-74.589,-178.247,10.154,149.552
C00859=1110.019,270.164,-74.619,-178.244,10.157,149.552
C00860=1110.015,270.412,-74.649,-178.240,10.159,149.552
C00861=1110.011,270.660,-74.678,-178.237,10.162,149.552
C00862=1110.007,270.908,-74.708,-178.235,10.164,149.552
C00863=1110.003,271.157,-74.738,-178.232,10.167,149.552
C00864=1109.998,271.405,-74.768,-178.229,10.169,149.551
C00865=1109.994,271.654,-74.798,-178.226,10.172,149.551
C00866=1109.990,271.901,-74.828,-178.223,10.175,149.551
C00867=1109.986,272.149,-74.858,-178.220,10.178,149.551
C00868=1109.981,272.398,-74.888,-178.218,10.180,149.551
C00869=1109.977,272.646,-74.918,-178.215,10.182,149.551
C00870=1109.973,272.894,-74.947,-178.212,10.185,149.551
C00871=1109.969,273.142,-74.977,-178.209,10.188,149.551
C00872=1109.964,273.390,-75.007,-178.206,10.191,149.551
C00873=1109.961,273.639,-75.037,-178.203,10.193,149.551
C00874=1109.957,273.887,-75.067,-178.200,10.196,149.550
C00875=1109.952,274.135,-75.097,-178.198,10.198,149.550
C00876=1109.948,274.383,-75.128,-178.195,10.201,149.550
C00877=1109.944,274.631,-75.157,-178.192,10.203,149.550
C00878=1109.939,274.879,-75.188,-178.189,10.206,149.550
C00879=1109.936,275.127,-75.218,-178.186,10.209,149.550
C00880=1109.932,275.376,-75.248,-178.183,10.212,149.550
C00881=1109.927,275.624,-75.279,-178.180,10.214,149.550
C00882=1109.923,275.872,-75.308,-178.178,10.216,149.549
C00883=1109.919,276.120,-75.338,-178.175,10.219,149.549
C00884=1109.914,276.368,-75.368,-178.172,10.222,149.549
C00885=1109.910,276.616,-75.398,-178.169,10.224,149.549
C00886=1109.907,276.864,-75.429,-178.166,10.227,149.549
C00887=1109.902,277.113,-75.459,-178.163,10.230,149.549
C00888=1109.898,277.361,-75.489,-178.160,10.233,149.549
C00889=1109.894,277.608,-75.520,-178.156,10.235,149.548
C00890=1109.890,277.857,-75.550,-178.154,10.238,149.548
C00891=1109.886,278.105,-75.581,-178.151,10.240,149.548
C00892=1109.882,278.353,-75.611,-178.148,10.243,149.548
C00893=1109.878,278.601,-75.641,-178.145,10.245,149.548
C00894=1109.873,278.849,-75.671,-178.142,10.248,149.548
C00895=1109.870,279.098,-75.701,-178.139,10.250,149.548
C00896=1109.865,279.346,-75.732,-178.136,10.253,149.548
C00897=1109.861,279.593,-75.762,-178.133,10.256,149.547
C00898=1109.856,279.842,-75.792,-178.130,10.258,149.547
C00899=1109.852,280.090,-75.824,-178.127,10.261,149.547
C00900=1109.848,280.338,-75.854,-178.124,10.263,149.547
C00901=1109.844,280.586,-75.884,-178.121,10.266,149.547
C00902=1109.840,280.834,-75.915,-178.118,10.268,149.547
C00903=1109.836,281.082,-75.946,-178.115,10.271,149.546
C00904=1109.832,281.330,-75.976,-178.112,10.273,149.546
C00905=1109.827,281.579,-76.006,-178.109,10.276,149.546
C00906=1109.824,281.791,-76.033,-178.106,10.278,149.546
C00907=1109.821,282.004,-76.058,-178.104,10.281,149.546
C00908=1109.816,282.216,-76.085,-178.101,10.283,149.546
C00909=1109.813,282.428,-76.111,-178.099,10.285,149.545
C00910=1109.809,282.640,-76.137,-178.096,10.287,149.545
C00911=1109.806,282.853,-76.164,-178.093,10.289,149.545
C00912=1109.803,283.065,-76.190,-178.091,10.291,149.545
C00913=1109.799,283.278,-76.215,-178.089,10.293,149.545
C00914=1109.795,283.526,-76.247,-178.085,10.295,149.545
C00915=1109.790,283.774,-76.277,-178.082,10.298,149.544
C00916=1109.786,284.022,-76.307,-178.079,10.301,149.544
C00917=1109.782,284.271,-76.339,-178.076,10.303,149.544
C00918=1109.778,284.518,-76.370,-178.073,10.306,149.544
C00919=1109.775,284.766,-76.401,-178.070,10.309,149.544
C00920=1109.770,285.014,-76.431,-178.067,10.311,149.544
C00921=1109.765,285.262,-76.462,-178.064,10.314,149.544
C00922=1109.762,285.510,-76.493,-178.061,10.316,149.543
C00923=1109.757,285.758,-76.523,-178.058,10.319,149.543
C00924=1109.753,286.006,-76.554,-178.055,10.321,149.543
C00925=1109.749,286.255,-76.585,-178.052,10.324,149.543
C00926=1109.745,286.502,-76.616,-178.049,10.326,149.543
C00927=1109.741,286.751,-76.647,-178.046,10.329,149.542
C00928=1109.737,286.999,-76.678,-178.043,10.332,149.542
C00929=1109.732,287.247,-76.709,-178.039,10.334,149.542
C00930=1109.729,287.495,-76.739,-178.037,10.336,149.542
C00931=1109.724,287.742,-76.771,-178.034,10.338,149.542
C00932=1109.720,287.991,-76.802,-178.031,10.341,149.542
C00933=1109.716,288.239,-76.833,-178.028,10.344,149.541
C00934=1109.712,288.488,-76.864,-178.025,10.346,149.541
C00935=1109.708,288.735,-76.895,-178.022,10.349,149.541
C00936=1109.704,288.983,-76.926,-178.018,10.352,149.541
C00937=1109.700,289.231,-76.957,-178.015,10.354,149.541
C00938=1109.695,289.479,-76.988,-178.013,10.356,149.540
C00939=1109.691,289.727,-77.019,-178.010,10.359,149.540
C00940=1109.687,289.975,-77.050,-178.006,10.361,149.540
C00941=1109.683,290.223,-77.082,-178.004,10.364,149.540
C00942=1109.679,290.471,-77.112,-178.000,10.366,149.540
C00943=1109.675,290.719,-77.144,-177.997,10.369,149.540
C00944=1109.671,290.967,-77.175,-177.994,10.372,149.540
C00945=1109.667,291.216,-77.206,-177.991,10.374,149.539
C00946=1109.662,291.463,-77.237,-177.988,10.377,149.539
C00947=1109.658,291.712,-77.268,-177.985,10.379,149.539
C00948=1109.654,291.959,-77.300,-177.982,10.382,149.539
C00949=1109.650,292.208,-77.331,-177.979,10.384,149.539
C00950=1109.646,292.455,-77.363,-177.976,10.387,149.538
C00951=1109.642,292.704,-77.394,-177.973,10.389,149.538
C00952=1109.638,292.952,-77.425,-177.970,10.392,149.538
C00953=1109.633,293.200,-77.456,-177.967,10.394,149.538
C00954=1109.630,293.448,-77.488,-177.964,10.397,149.538
C00955=1109.625,293.695,-77.520,-177.961,10.399,149.538
C00956=1109.621,293.944,-77.551,-177.958,10.402,149.537
C00957=1109.617,294.191,-77.582,-177.955,10.404,149.537
C00958=1109.613,294.440,-77.613,-177.952,10.407,149.537
C00959=1109.609,294.687,-77.645,-177.949,10.409,149.537
C00960=1109.605,294.935,-77.677,-177.945,10.412,149.537
C00961=1109.601,295.184,-77.708,-177.942,10.415,149.537
C00962=1109.598,295.396,-77.734,-177.940,10.417,149.536
C00963=1109.594,295.608,-77.761,-177.937,10.418,149.536
C00964=1109.590,295.820,-77.788,-177.935,10.421,149.536
C00965=1109.587,296.032,-77.815,-177.932,10.423,149.536
C00966=1109.584,296.245,-77.842,-177.930,10.425,149.536
C00967=1109.580,296.457,-77.870,-177.927,10.428,149.536
C00968=1109.577,296.669,-77.897,-177.924,10.430,149.536
C00969=1109.574,296.881,-77.924,-177.922,10.431,149.535
C00970=1109.569,297.129,-77.955,-177.919,10.434,149.535
C00971=1109.565,297.377,-77.987,-177.916,10.437,149.535
C00972=1109.562,297.625,-78.018,-177.912,10.439,149.535
C00973=1109.556,297.873,-78.051,-177.909,10.442,149.535
C00974=1109.553,298.121,-78.082,-177.906,10.444,149.534
C00975=1109.549,298.369,-78.114,-177.903,10.447,149.534
C00976=1109.544,298.617,-78.145,-177.900,10.450,149.534
C00977=1109.541,298.865,-78.177,-177.898,10.452,149.534
C00978=1109.536,299.113,-78.209,-177.894,10.454,149.534
C00979=1109.532,299.361,-78.241,-177.891,10.457,149.534
C00980=1109.528,299.609,-78.273,-177.888,10.459,149.533
C00981=1109.525,299.857,-78.304,-177.885,10.462,149.533
C00982=1109.520,300.104,-78.336,-177.882,10.464,149.533
C00983=1109.516,300.352,-78.368,-177.879,10.467,149.533
C00984=1109.512,300.600,-78.400,-177.875,10.470,149.533
C00985=1109.508,300.848,-78.432,-177.873,10.472,149.533
C00986=1109.504,301.096,-78.464,-177.870,10.474,149.532
C00987=1109.500,301.344,-78.496,-177.867,10.477,149.532
C00988=1109.495,301.591,-78.527,-177.864,10.479,149.532
C00989=1109.492,301.839,-78.559,-177.861,10.482,149.532
C00990=1109.487,302.088,-78.592,-177.857,10.484,149.532
C00991=1109.483,302.336,-78.624,-177.854,10.487,149.532
C00992=1109.479,302.583,-78.655,-177.851,10.490,149.531
C00993=1109.475,302.832,-78.687,-177.848,10.492,149.531
C00994=1109.471,303.080,-78.719,-177.845,10.495,149.531
C00995=1109.467,303.327,-78.751,-177.842,10.497,149.531
C00996=1109.462,303.575,-78.783,-177.839,10.499,149.531
C00997=1109.459,303.823,-78.815,-177.836,10.502,149.531
C00998=1109.455,304.071,-78.848,-177.833,10.504,149.530
C00999=1109.451,304.319,-78.880,-177.830,10.507,149.530
C01000=1109.446,304.566,-78.912,-177.827,10.510,149.530
C01001=1109.442,304.815,-78.944,-177.824,10.512,149.530
C01002=1109.438,305.063,-78.976,-177.820,10.515,149.530
C01003=1109.434,305.311,-79.008,-177.817,10.518,149.529
C01004=1109.430,305.558,-79.040,-177.815,10.519,149.529
C01005=1109.426,305.806,-79.072,-177.812,10.522,149.529
C01006=1109.422,306.054,-79.105,-177.808,10.524,149.529
C01007=1109.418,306.302,-79.137,-177.806,10.527,149.529
C01008=1109.414,306.550,-79.170,-177.802,10.530,149.529
C01009=1109.410,306.798,-79.202,-177.799,10.532,149.528
C01010=1109.405,307.046,-79.234,-177.796,10.535,149.528
C01011=1109.402,307.293,-79.266,-177.793,10.538,149.528
C01012=1109.397,307.542,-79.299,-177.790,10.540,149.528
C01013=1109.394,307.790,-79.331,-177.786,10.543,149.528
C01014=1109.389,308.037,-79.364,-177.784,10.544,149.527
C01015=1109.386,308.285,-79.396,-177.781,10.547,149.527
C01016=1109.382,308.533,-79.429,-177.778,10.550,149.527
C01017=1109.377,308.780,-79.460,-177.774,10.552,149.527
C01018=1109.374,308.992,-79.488,-177.772,10.554,149.527
C01019=1109.371,309.205,-79.516,-177.769,10.557,149.527
C01020=1109.367,309.417,-79.544,-177.767,10.559,149.526
C01021=1109.363,309.629,-79.572,-177.764,10.561,149.526
C01022=1109.360,309.841,-79.600,-177.761,10.563,149.526
C01023=1109.356,310.054,-79.627,-177.759,10.565,149.526
C01024=1109.353,310.266,-79.655,-177.756,10.567,149.526
C01025=1109.349,310.477,-79.683,-177.753,10.570,149.526
C01026=1109.346,310.726,-79.715,-177.750,10.572,149.526
C01027=1109.342,310.973,-79.748,-177.747,10.575,149.525
C01028=1109.337,311.221,-79.781,-177.744,10.577,149.525
C01029=1109.334,311.469,-79.813,-177.741,10.579,149.525
C01030=1109.330,311.717,-79.846,-177.738,10.582,149.525
C01031=1109.325,311.965,-79.879,-177.735,10.584,149.525
C01032=1109.322,312.213,-79.911,-177.732,10.587,149.525
C01033=1109.318,312.460,-79.944,-177.729,10.590,149.524
C01034=1109.313,312.709,-79.977,-177.726,10.592,149.524
C01035=1109.310,312.956,-80.009,-177.722,10.595,149.524
C01036=1109.306,313.204,-80.043,-177.719,10.598,149.524
C01037=1109.301,313.452,-80.075,-177.717,10.599,149.524
C01038=1109.298,313.700,-80.108,-177.713,10.602,149.523
C01039=1109.293,313.947,-80.140,-177.711,10.604,149.523
C01040=1109.289,314.195,-80.173,-177.707,10.607,149.523
C01041=1109.285,314.442,-80.205,-177.704,10.610,149.523
C01042=1109.282,314.691,-80.239,-177.701,10.612,149.523
C01043=1109.278,314.938,-80.272,-177.698,10.615,149.523
C01044=1109.273,315.187,-80.304,-177.695,10.617,149.522
C01045=1109.270,315.434,-80.337,-177.691,10.620,149.522
C01046=1109.266,315.682,-80.370,-177.689,10.622,149.522
C01047=1109.261,315.930,-80.403,-177.686,10.624,149.522
C01048=1109.257,316.177,-80.437,-177.683,10.627,149.522
C01049=1109.253,316.425,-80.470,-177.679,10.629,149.521
C01050=1109.249,316.673,-80.502,-177.676,10.632,149.521
C01051=1109.245,316.921,-80.535,-177.673,10.635,149.521
C01052=1109.241,317.169,-80.568,-177.670,10.637,149.521
C01053=1109.237,317.416,-80.601,-177.667,10.640,149.521
C01054=1109.233,317.664,-80.634,-177.664,10.642,149.521
C01055=1109.229,317.912,-80.667,-177.660,10.645,149.520
C01056=1109.225,318.159,-80.700,-177.658,10.647,149.520
C01057=1109.221,318.407,-80.733,-177.655,10.649,149.520
C01058=1109.217,318.655,-80.766,-177.652,10.652,149.520
C01059=1109.214,318.903,-80.800,-177.648,10.654,149.520
C01060=1109.209,319.151,-80.833,-177.645,10.657,149.519
C01061=1109.205,319.399,-80.866,-177.642,10.660,149.519
C01062=1109.201,319.646,-80.899,-177.639,10.662,149.519
C01063=1109.198,319.894,-80.932,-177.636,10.665,149.519
C01064=1109.194,320.141,-80.965,-177.633,10.667,149.519
C01065=1109.189,320.389,-80.998,-177.630,10.669,149.519
C01066=1109.185,320.637,-81.031,-177.627,10.672,149.518
C01067=1109.182,320.885,-81.065,-177.624,10.674,149.518
C01068=1109.178,321.132,-81.099,-177.621,10.677,149.518
C01069=1109.174,321.380,-81.132,-177.617,10.679,149.518
C01070=1109.170,321.628,-81.165,-177.614,10.682,149.518
C01071=1109.166,321.876,-81.198,-177.611,10.685,149.518
C01072=1109.161,322.123,-81.231,-177.608,10.687,149.517
C01073=1109.158,322.372,-81.265,-177.605,10.689,149.517
C01074=1109.155,322.583,-81.293,-177.602,10.691,149.517
C01075=1109.151,322.795,-81.322,-177.600,10.693,149.517
C01076=1109.148,323.007,-81.351,-177.597,10.696,149.517
C01077=1109.144,323.219,-81.379,-177.594,10.698,149.517
C01078=1109.141,323.431,-81.407,-177.592,10.700,149.516
C01079=1109.137,323.643,-81.437,-177.589,10.702,149.516
C01080=1109.134,323.855,-81.465,-177.586,10.704,149.516
C01081=1109.130,324.067,-81.494,-177.584,10.706,149.516
C01082=1109.126,324.315,-81.527,-177.581,10.709,149.516
C01083=1109.123,324.563,-81.561,-177.578,10.711,149.516
C01084=1109.119,324.810,-81.595,-177.574,10.714,149.515
C01085=1109.115,325.058,-81.628,-177.571,10.716,149.515
C01086=1109.110,325.306,-81.661,-177.568,10.719,149.515
C01087=1109.107,325.553,-81.695,-177.565,10.721,149.515
C01088=1109.103,325.801,-81.728,-177.562,10.724,149.515
C01089=1109.099,326.049,-81.761,-177.559,10.726,149.514
C01090=1109.094,326.296,-81.796,-177.556,10.728,149.514
C01091=1109.091,326.545,-81.829,-177.553,10.731,149.514
C01092=1109.087,326.792,-81.863,-177.549,10.733,149.514
C01093=1109.083,327.040,-81.896,-177.546,10.736,149.514
C01094=1109.079,327.287,-81.930,-177.543,10.739,149.514
C01095=1109.076,327.535,-81.964,-177.540,10.741,149.513
C01096=1109.071,327.783,-81.998,-177.537,10.744,149.513
C01097=1109.067,328.030,-82.032,-177.534,10.746,149.513
C01098=1109.064,328.278,-82.066,-177.530,10.749,149.513
C01099=1109.059,328.526,-82.099,-177.528,10.750,149.512
C01100=1109.055,328.773,-82.133,-177.525,10.753,149.512
C01101=1109.051,329.021,-82.167,-177.521,10.756,149.512
C01102=1109.048,329.269,-82.201,-177.518,10.758,149.512
C01103=1109.044,329.516,-82.235,-177.515,10.761,149.512
C01104=1109.039,329.764,-82.268,-177.512,10.763,149.512
C01105=1109.036,330.012,-82.303,-177.508,10.766,149.511
C01106=1109.031,330.259,-82.336,-177.506,10.769,149.511
C01107=1109.027,330.507,-82.370,-177.502,10.771,149.511
C01108=1109.024,330.755,-82.404,-177.500,10.773,149.511
C01109=1109.020,331.002,-82.438,-177.497,10.776,149.511
C01110=1109.016,331.250,-82.472,-177.493,10.778,149.511
C01111=1109.012,331.498,-82.506,-177.490,10.780,149.510
C01112=1109.008,331.745,-82.540,-177.487,10.783,149.510
C01113=1109.004,331.993,-82.574,-177.484,10.786,149.510
C01114=1109.000,332.241,-82.608,-177.480,10.788,149.510
C01115=1108.996,332.488,-82.642,-177.477,10.791,149.510
C01116=1108.992,332.736,-82.677,-177.474,10.793,149.509
C01117=1108.988,332.984,-82.710,-177.471,10.796,149.509
C01118=1108.985,333.231,-82.744,-177.468,10.797,149.509
C01119=1108.980,333.479,-82.779,-177.465,10.800,149.509
C01120=1108.976,333.726,-82.813,-177.462,10.803,149.509
C01121=1108.972,333.974,-82.847,-177.459,10.805,149.508
C01122=1108.968,334.221,-82.881,-177.455,10.808,149.508
C01123=1108.965,334.469,-82.916,-177.452,10.810,149.508
C01124=1108.960,334.717,-82.949,-177.449,10.813,149.508
C01125=1108.957,334.965,-82.984,-177.446,10.815,149.508
C01126=1108.952,335.212,-83.018,-177.443,10.818,149.508
C01127=1108.949,335.460,-83.052,-177.440,10.820,149.507
C01128=1108.945,335.707,-83.087,-177.437,10.822,149.507
C01129=1108.941,335.955,-83.121,-177.434,10.825,149.507
C01130=1108.935,336.362,-83.177,-177.428,10.829,149.507
C01131=1108.929,336.770,-83.234,-177.423,10.833,149.506
C01132=1108.922,337.178,-83.290,-177.418,10.837,149.506
C01133=1108.915,337.586,-83.348,-177.413,10.841,149.506
C01134=1108.911,337.833,-83.382,-177.409,10.844,149.505
C01135=1108.908,338.081,-83.416,-177.406,10.846,149.505
C01136=1108.904,338.328,-83.450,-177.403,10.849,149.505
C01137=1108.900,338.576,-83.485,-177.401,10.851,149.505
C01138=1108.895,338.823,-83.520,-177.397,10.853,149.505
C01139=1108.892,339.071,-83.554,-177.394,10.856,149.504
C01140=1108.888,339.318,-83.589,-177.391,10.858,149.504
C01141=1108.884,339.566,-83.623,-177.388,10.861,149.504
C01142=1108.880,339.813,-83.658,-177.384,10.863,149.504
C01143=1108.876,340.062,-83.692,-177.381,10.866,149.504
C01144=1108.872,340.308,-83.727,-177.378,10.869,149.504
C01145=1108.868,340.556,-83.762,-177.375,10.871,149.503
C01146=1108.864,340.804,-83.796,-177.372,10.873,149.503
C01147=1108.861,341.051,-83.831,-177.369,10.875,149.503
C01148=1108.856,341.298,-83.866,-177.366,10.878,149.503
C01149=1108.852,341.546,-83.901,-177.363,10.880,149.503
C01150=1108.848,341.794,-83.935,-177.359,10.883,149.502
C01151=1108.845,342.042,-83.969,-177.356,10.885,149.502
C01152=1108.841,342.289,-84.005,-177.353,10.888,149.502
C01153=1108.836,342.536,-84.039,-177.350,10.891,149.502
C01154=1108.589,331.704,-82.594,-177.487,10.783,149.510
C01155=1108.593,331.457,-82.560,-177.490,10.780,149.510
C01156=1108.597,331.209,-82.525,-177.493,10.778,149.511
C01157=1108.601,330.962,-82.492,-177.496,10.776,149.511
C01158=1108.605,330.714,-82.458,-177.499,10.774,149.511
C01159=1108.608,330.466,-82.424,-177.502,10.771,149.511
C01160=1108.612,330.219,-82.390,-177.505,10.768,149.511
C01161=1108.617,329.971,-82.357,-177.508,10.766,149.511
C01162=1108.620,329.723,-82.322,-177.512,10.763,149.512
C01163=1108.625,329.475,-82.289,-177.515,10.761,149.512
C01164=1108.629,329.228,-82.255,-177.518,10.758,149.512
C01165=1108.632,328.981,-82.220,-177.521,10.756,149.512
C01166=1108.636,328.733,-82.187,-177.524,10.754,149.512
C01167=1108.640,328.485,-82.153,-177.527,10.751,149.513
C01168=1108.644,328.237,-82.119,-177.530,10.749,149.513
C01169=1108.648,327.990,-82.085,-177.533,10.746,149.513
C01170=1108.652,327.742,-82.052,-177.537,10.744,149.513
C01171=1108.656,327.494,-82.017,-177.540,10.741,149.513
C01172=1108.660,327.246,-81.984,-177.543,10.738,149.513
C01173=1108.664,326.999,-81.950,-177.546,10.736,149.514
C01174=1108.668,326.751,-81.917,-177.549,10.733,149.514
C01175=1108.671,326.504,-81.883,-177.552,10.731,149.514
C01176=1108.675,326.256,-81.850,-177.555,10.729,149.514
C01177=1108.680,326.008,-81.815,-177.558,10.727,149.514
C01178=1108.684,325.761,-81.782,-177.561,10.724,149.514
C01179=1108.688,325.512,-81.749,-177.565,10.721,149.515
C01180=1108.692,325.265,-81.715,-177.568,10.719,149.515
C01181=1108.696,325.017,-81.682,-177.571,10.716,149.515
C01182=1108.700,324.770,-81.649,-177.574,10.714,149.515
C01183=1108.703,324.522,-81.614,-177.578,10.711,149.516
C01184=1108.707,324.274,-81.581,-177.580,10.708,149.516
C01185=1108.711,324.026,-81.548,-177.583,10.707,149.516
C01186=1108.715,323.779,-81.514,-177.586,10.704,149.516
C01187=1108.722,323.427,-81.467,-177.591,10.700,149.516
C01188=1108.726,323.076,-81.419,-177.595,10.697,149.517
C01189=1108.732,322.724,-81.371,-177.600,10.693,149.517
C01190=1108.738,322.373,-81.324,-177.604,10.690,149.517
C01191=1108.742,322.125,-81.291,-177.607,10.687,149.517
C01192=1108.746,321.878,-81.257,-177.610,10.685,149.517
C01193=1108.750,321.629,-81.224,-177.613,10.683,149.518
C01194=1108.754,321.382,-81.191,-177.616,10.680,149.518
C01195=1108.758,321.134,-81.157,-177.620,10.677,149.518
C01196=1108.762,320.886,-81.124,-177.623,10.675,149.518
C01197=1108.766,320.639,-81.091,-177.626,10.672,149.518
C01198=1108.770,320.391,-81.058,-177.629,10.670,149.519
C01199=1108.774,320.142,-81.024,-177.632,10.668,149.519
C01200=1108.777,319.896,-80.991,-177.635,10.665,149.519
C01201=1108.781,319.648,-80.958,-177.638,10.663,149.519
C01202=1108.785,319.400,-80.925,-177.641,10.660,149.519
C01203=1108.789,319.152,-80.892,-177.644,10.658,149.519
C01204=1108.794,318.905,-80.859,-177.647,10.655,149.520
C01205=1108.798,318.657,-80.825,-177.651,10.652,149.520
C01206=1108.802,318.409,-80.792,-177.654,10.650,149.520
C01207=1108.805,318.161,-80.759,-177.657,10.647,149.520
C01208=1108.809,317.913,-80.726,-177.660,10.645,149.520
C01209=1108.813,317.666,-80.693,-177.663,10.643,149.520
C01210=1108.817,317.417,-80.661,-177.666,10.640,149.521
C01211=1108.821,317.170,-80.627,-177.669,10.638,149.521
C01212=1108.826,316.922,-80.594,-177.672,10.635,149.521
C01213=1108.830,316.674,-80.561,-177.676,10.633,149.521
C01214=1108.833,316.427,-80.529,-177.678,10.630,149.521
C01215=1108.837,316.179,-80.495,-177.682,10.627,149.522
C01216=1108.841,315.931,-80.462,-177.685,10.625,149.522
C01217=1108.846,315.683,-80.429,-177.688,10.622,149.522
C01218=1108.850,315.435,-80.397,-177.691,10.620,149.522
C01219=1108.853,315.188,-80.364,-177.694,10.618,149.522
C01220=1108.858,314.940,-80.331,-177.697,10.615,149.522
C01221=1108.862,314.692,-80.298,-177.700,10.612,149.523
C01222=1108.866,314.445,-80.265,-177.703,10.610,149.523
C01223=1108.869,314.196,-80.233,-177.707,10.608,149.523
C01224=1108.874,313.949,-80.200,-177.709,10.605,149.523
C01225=1108.878,313.701,-80.166,-177.713,10.602,149.523
C01226=1108.881,313.453,-80.135,-177.716,10.600,149.523
C01227=1108.886,313.205,-80.101,-177.718,10.598,149.524
C01228=1108.890,312.958,-80.068,-177.721,10.595,149.524
C01229=1108.893,312.709,-80.036,-177.725,10.593,149.524
C01230=1108.898,312.462,-80.003,-177.728,10.590,149.524
C01231=1108.902,312.214,-79.970,-177.731,10.588,149.524
C01232=1108.905,311.966,-79.938,-177.734,10.585,149.525
C01233=1108.910,311.718,-79.905,-177.737,10.582,149.525
C01234=1108.914,311.471,-79.872,-177.741,10.580,149.525
C01235=1108.917,311.222,-79.840,-177.743,10.577,149.525
C01236=1108.922,310.975,-79.807,-177.747,10.575,149.525
C01237=1108.926,310.726,-79.775,-177.749,10.573,149.525
C01238=1108.929,310.479,-79.742,-177.752,10.570,149.526
C01239=1108.933,310.267,-79.714,-177.755,10.567,149.526
C01240=1108.936,310.055,-79.687,-177.758,10.566,149.526
C01241=1108.940,309.843,-79.659,-177.760,10.564,149.526
C01242=1108.943,309.631,-79.631,-177.763,10.561,149.526
C01243=1108.947,309.419,-79.603,-177.766,10.559,149.526
C01244=1108.951,309.206,-79.575,-177.768,10.557,149.527
C01245=1108.954,308.994,-79.547,-177.771,10.555,149.527
C01246=1108.958,308.783,-79.519,-177.774,10.553,149.527
C01247=1108.962,308.535,-79.488,-177.777,10.550,149.527
C01248=1108.966,308.287,-79.454,-177.780,10.548,149.527
C01249=1108.969,308.039,-79.423,-177.783,10.545,149.527
C01250=1108.974,307.790,-79.390,-177.786,10.543,149.528
C01251=1108.977,307.543,-79.358,-177.789,10.541,149.528
C01252=1108.982,307.295,-79.326,-177.792,10.538,149.528
C01253=1108.986,307.047,-79.294,-177.795,10.535,149.528
C01254=1108.990,306.800,-79.261,-177.798,10.533,149.528
C01255=1108.994,306.552,-79.229,-177.801,10.530,149.528
C01256=1108.998,306.303,-79.196,-177.805,10.528,149.529
C01257=1109.002,306.056,-79.164,-177.807,10.525,149.529
C01258=1109.007,305.808,-79.132,-177.811,10.522,149.529
C01259=1109.010,305.560,-79.100,-177.814,10.520,149.529
C01260=1109.014,305.312,-79.068,-177.816,10.518,149.529
C01261=1109.018,305.064,-79.035,-177.820,10.516,149.530
C01262=1109.022,304.816,-79.003,-177.823,10.513,149.530
C01263=1109.027,304.569,-78.971,-177.826,10.510,149.530
C01264=1109.031,304.321,-78.939,-177.829,10.508,149.530
C01265=1109.034,304.073,-78.907,-177.832,10.505,149.530
C01266=1109.039,303.825,-78.874,-177.835,10.502,149.530
C01267=1109.043,303.577,-78.843,-177.839,10.500,149.531
C01268=1109.047,303.329,-78.810,-177.841,10.497,149.531
C01269=1109.051,303.081,-78.778,-177.844,10.496,149.531
C01270=1109.055,302.833,-78.746,-177.847,10.493,149.531
C01271=1109.060,302.585,-78.714,-177.850,10.490,149.531
C01272=1109.063,302.337,-78.682,-177.853,10.488,149.531
C01273=1109.067,302.089,-78.651,-177.857,10.485,149.532
C01274=1109.072,301.841,-78.618,-177.860,10.482,149.532
C01275=1109.076,301.594,-78.587,-177.863,10.480,149.532
C01276=1109.080,301.346,-78.555,-177.866,10.477,149.532
C01277=1109.084,301.097,-78.522,-177.869,10.475,149.532
C01278=1109.088,300.850,-78.491,-177.871,10.473,149.532
C01279=1109.092,300.602,-78.459,-177.875,10.470,149.533
C01280=1109.096,300.354,-78.427,-177.878,10.468,149.533
C01281=1109.100,300.105,-78.395,-177.881,10.465,149.533
C01282=1109.105,299.858,-78.363,-177.884,10.462,149.533
C01283=1109.108,299.610,-78.331,-177.887,10.460,149.533
C01284=1109.112,299.362,-78.300,-177.890,10.457,149.533
C01285=1109.117,299.114,-78.268,-177.894,10.455,149.534
C01286=1109.121,298.866,-78.236,-177.897,10.452,149.534
C01287=1109.124,298.618,-78.204,-177.899,10.450,149.534
C01288=1109.129,298.370,-78.173,-177.902,10.448,149.534
C01289=1109.133,298.122,-78.141,-177.906,10.445,149.534
C01290=1109.136,297.874,-78.109,-177.908,10.442,149.535
C01291=1109.141,297.627,-78.077,-177.912,10.440,149.535
C01292=1109.145,297.379,-78.046,-177.915,10.437,149.535
C01293=1109.149,297.131,-78.014,-177.918,10.435,149.535
C01294=1109.153,296.883,-77.983,-177.921,10.432,149.535
C01295=1109.157,296.670,-77.956,-177.923,10.430,149.535
C01296=1109.160,296.458,-77.929,-177.926,10.428,149.536
C01297=1109.164,296.246,-77.901,-177.929,10.426,149.536
C01298=1109.167,296.034,-77.874,-177.931,10.424,149.536
C01299=1109.171,295.822,-77.848,-177.934,10.422,149.536
C01300=1109.174,295.610,-77.820,-177.937,10.419,149.536
C01301=1109.178,295.397,-77.793,-177.939,10.417,149.536
C01302=1109.181,295.185,-77.767,-177.941,10.415,149.536
C01303=1109.185,294.936,-77.736,-177.945,10.413,149.537
C01304=1109.189,294.689,-77.704,-177.948,10.410,149.537
C01305=1109.193,294.441,-77.672,-177.951,10.407,149.537
C01306=1109.198,294.193,-77.641,-177.954,10.405,149.537
C01307=1109.201,293.945,-77.610,-177.957,10.402,149.537
C01308=1109.206,293.698,-77.578,-177.960,10.400,149.537
C01309=1109.210,293.449,-77.547,-177.963,10.398,149.538
C01310=1109.213,293.201,-77.515,-177.966,10.395,149.538
C01311=1109.218,292.953,-77.484,-177.969,10.392,149.538
C01312=1109.222,292.705,-77.453,-177.972,10.390,149.538
C01313=1109.226,292.457,-77.422,-177.975,10.387,149.538
C01314=1109.230,292.209,-77.390,-177.978,10.385,149.539
C01315=1109.235,291.961,-77.359,-177.981,10.382,149.539
C01316=1109.238,291.713,-77.327,-177.984,10.379,149.539
C01317=1109.243,291.465,-77.297,-177.987,10.378,149.539
C01318=1109.247,291.217,-77.265,-177.990,10.375,149.539
C01319=1109.251,290.969,-77.234,-177.993,10.372,149.539
C01320=1109.255,290.721,-77.202,-177.996,10.370,149.540
C01321=1109.260,290.473,-77.171,-178.000,10.367,149.540
C01322=1109.264,290.224,-77.140,-178.002,10.364,149.540
C01323=1109.267,289.977,-77.109,-178.006,10.362,149.540
C01324=1109.271,289.729,-77.078,-178.009,10.359,149.540
C01325=1109.276,289.481,-77.047,-178.012,10.356,149.540
C01326=1109.280,289.233,-77.016,-178.014,10.355,149.541
C01327=1109.284,288.985,-76.985,-178.017,10.352,149.541
C01328=1109.288,288.737,-76.953,-178.021,10.350,149.541
C01329=1109.292,288.489,-76.923,-178.024,10.347,149.541
C01330=1109.296,288.240,-76.892,-178.027,10.344,149.541
C01331=1109.300,287.992,-76.861,-178.030,10.342,149.541
C01332=1109.305,287.745,-76.829,-178.033,10.339,149.542
C01333=1109.309,287.496,-76.798,-178.036,10.336,149.542
C01334=1109.313,287.249,-76.768,-178.038,10.334,149.542
C01335=1109.317,287.000,-76.737,-178.042,10.332,149.542
C01336=1109.321,286.753,-76.706,-178.045,10.329,149.542
C01337=1109.325,286.504,-76.674,-178.048,10.327,149.543
C01338=1109.329,286.257,-76.644,-178.051,10.324,149.543
C01339=1109.333,286.009,-76.613,-178.054,10.322,149.543
C01340=1109.337,285.760,-76.582,-178.057,10.319,149.543
C01341=1109.342,285.512,-76.552,-178.060,10.316,149.543
C01342=1109.346,285.264,-76.521,-178.063,10.315,149.543
C01343=1109.350,285.016,-76.490,-178.066,10.312,149.543
C01344=1109.354,284.768,-76.459,-178.069,10.309,149.544
C01345=1109.358,284.520,-76.428,-178.072,10.307,149.544
C01346=1109.362,284.272,-76.398,-178.075,10.304,149.544
C01347=1109.367,284.024,-76.367,-178.078,10.301,149.544
C01348=1109.371,283.775,-76.336,-178.081,10.299,149.544
C01349=1109.375,283.528,-76.305,-178.085,10.296,149.545
C01350=1109.379,283.280,-76.275,-178.087,10.294,149.545
C01351=1109.382,283.067,-76.249,-178.090,10.291,149.545
C01352=1109.385,282.855,-76.222,-178.093,10.290,149.545
C01353=1109.390,282.642,-76.196,-178.095,10.288,149.545
C01354=1109.393,282.430,-76.169,-178.098,10.285,149.545
C01355=1109.397,282.218,-76.144,-178.100,10.283,149.545
C01356=1109.401,282.005,-76.117,-178.102,10.281,149.546
C01357=1109.404,281.793,-76.091,-178.106,10.279,149.546
C01358=1109.408,281.581,-76.065,-178.108,10.277,149.546
C01359=1109.412,281.332,-76.034,-178.111,10.274,149.546
C01360=1109.416,281.084,-76.004,-178.114,10.272,149.546
C01361=1109.420,280.837,-75.973,-178.117,10.269,149.546
C01362=1109.424,280.589,-75.943,-178.120,10.266,149.547
C01363=1109.428,280.340,-75.913,-178.123,10.264,149.547
C01364=1109.433,280.092,-75.882,-178.126,10.262,149.547
C01365=1109.437,279.844,-75.852,-178.129,10.259,149.547
C01366=1109.441,279.596,-75.821,-178.132,10.256,149.547
C01367=1109.445,279.348,-75.790,-178.135,10.254,149.547
C01368=1109.450,279.099,-75.760,-178.138,10.251,149.547
C01369=1109.454,278.851,-75.730,-178.141,10.248,149.548
C01370=1109.458,278.604,-75.699,-178.144,10.246,149.548
C01371=1109.461,278.355,-75.669,-178.147,10.244,149.548
C01372=1109.466,278.107,-75.639,-178.150,10.241,149.548
C01373=1109.470,277.859,-75.609,-178.153,10.238,149.548
C01374=1109.474,277.611,-75.578,-178.156,10.236,149.548
C01375=1109.478,277.363,-75.547,-178.159,10.233,149.549
C01376=1109.482,277.114,-75.518,-178.162,10.230,149.549
C01377=1109.487,276.866,-75.487,-178.165,10.227,149.549
C01378=1109.491,276.618,-75.458,-178.168,10.225,149.549
C01379=1109.495,276.370,-75.428,-178.170,10.223,149.549
C01380=1109.499,276.122,-75.396,-178.173,10.220,149.549
C01381=1109.503,275.874,-75.367,-178.176,10.218,149.549
C01382=1109.508,275.626,-75.336,-178.179,10.215,149.549
C01383=1109.512,275.377,-75.307,-178.182,10.212,149.550
C01384=1109.516,275.130,-75.277,-178.185,10.209,149.550
C01385=1109.520,274.882,-75.246,-178.188,10.206,149.550
C01386=1109.524,274.633,-75.216,-178.191,10.204,149.550
C01387=1109.528,274.385,-75.186,-178.194,10.202,149.550
C01388=1109.533,274.137,-75.156,-178.197,10.199,149.550
C01389=1109.537,273.889,-75.126,-178.199,10.197,149.550
C01390=1109.541,273.641,-75.096,-178.202,10.194,149.550
C01391=1109.545,273.393,-75.066,-178.205,10.191,149.550
C01392=1109.550,273.144,-75.036,-178.208,10.188,149.551
C01393=1109.554,272.897,-75.006,-178.211,10.186,149.551
C01394=1109.557,272.648,-74.976,-178.214,10.184,149.551
C01395=1109.562,272.399,-74.946,-178.216,10.181,149.551
C01396=1109.566,272.152,-74.916,-178.219,10.178,149.551
C01397=1109.570,271.903,-74.886,-178.222,10.175,149.551
C01398=1109.574,271.656,-74.856,-178.225,10.172,149.551
C01399=1109.578,271.407,-74.827,-178.228,10.170,149.551
C01400=1109.583,271.159,-74.797,-178.230,10.168,149.551
C01401=1109.587,270.911,-74.766,-178.233,10.165,149.552
C01402=1109.591,270.663,-74.737,-178.237,10.163,149.552
C01403=1109.595,270.415,-74.708,-178.240,10.160,149.552
C01404=1109.600,270.166,-74.677,-178.243,10.157,149.552
C01405=1109.604,269.918,-74.647,-178.246,10.154,149.552
C01406=1109.608,269.670,-74.618,-178.248,10.152,149.552
C01407=1109.612,269.457,-74.592,-178.251,10.150,149.552
C01408=1109.615,269.245,-74.566,-178.253,10.147,149.552
C01409=1109.619,269.032,-74.541,-178.255,10.145,149.552
C01410=1109.622,268.820,-74.516,-178.257,10.143,149.552
C01411=1109.625,268.607,-74.490,-178.260,10.140,149.553
C01412=1109.629,268.395,-74.466,-178.263,10.139,149.553
C01413=1109.633,268.182,-74.440,-178.265,10.137,149.553
C01414=1109.637,267.970,-74.414,-178.267,10.135,149.553
C01415=1109.641,267.721,-74.385,-178.270,10.132,149.553
C01416=1109.645,267.473,-74.355,-178.273,10.129,149.553
C01417=1109.649,267.225,-74.326,-178.276,10.126,149.553
C01418=1109.653,266.977,-74.296,-178.278,10.124,149.553
C01419=1109.657,266.729,-74.266,-178.281,10.122,149.553
C01420=1109.662,266.480,-74.236,-178.284,10.119,149.554
C01421=1109.666,266.232,-74.207,-178.287,10.116,149.554
C01422=1109.670,265.984,-74.177,-178.289,10.114,149.554
C01423=1109.675,265.736,-74.148,-178.292,10.111,149.554
C01424=1109.679,265.487,-74.118,-178.296,10.109,149.554
C01425=1109.683,265.239,-74.089,-178.299,10.106,149.554
C01426=1109.688,264.991,-74.060,-178.301,10.104,149.554
C01427=1109.692,264.743,-74.030,-178.304,10.101,149.555
C01428=1109.696,264.495,-74.001,-178.307,10.099,149.555
C01429=1109.700,264.247,-73.971,-178.310,10.096,149.555
C01430=1109.705,263.998,-73.942,-178.313,10.093,149.555
C01431=1109.709,263.750,-73.913,-178.316,10.091,149.555
C01432=1109.713,263.502,-73.883,-178.318,10.089,149.555
C01433=1109.717,263.254,-73.854,-178.321,10.086,149.555
C01434=1109.721,263.005,-73.824,-178.324,10.083,149.555
C01435=1109.726,262.756,-73.795,-178.327,10.080,149.556
C01436=1109.730,262.508,-73.766,-178.330,10.078,149.556
C01437=1109.734,262.261,-73.737,-178.333,10.075,149.556
C01438=1109.738,262.013,-73.708,-178.336,10.072,149.556
C01439=1109.742,261.764,-73.679,-178.339,10.069,149.556
C01440=1109.747,261.516,-73.649,-178.342,10.067,149.556
C01441=1109.751,261.267,-73.620,-178.345,10.064,149.556
C01442=1109.755,261.019,-73.591,-178.347,10.062,149.556
C01443=1109.759,260.771,-73.561,-178.350,10.059,149.556
C01444=1109.764,260.523,-73.532,-178.353,10.056,149.557
C01445=1109.768,260.275,-73.503,-178.356,10.054,149.557
C01446=1109.772,260.026,-73.475,-178.359,10.051,149.557
C01447=1109.776,259.778,-73.445,-178.361,10.048,149.557
C01448=1109.780,259.530,-73.416,-178.364,10.045,149.557
C01449=1109.785,259.281,-73.387,-178.367,10.042,149.557
C01450=1109.790,259.033,-73.358,-178.370,10.039,149.557
C01451=1109.793,258.785,-73.329,-178.373,10.037,149.557
C01452=1109.797,258.537,-73.300,-178.375,10.034,149.557
C01453=1109.802,258.288,-73.271,-178.378,10.032,149.557
C01454=1109.806,258.040,-73.242,-178.381,10.029,149.557
C01455=1109.810,257.792,-73.214,-178.384,10.026,149.557
C01456=1109.815,257.544,-73.184,-178.386,10.023,149.557
C01457=1109.819,257.296,-73.155,-178.389,10.020,149.557
C01458=1109.823,257.047,-73.126,-178.392,10.017,149.557
C01459=1109.827,256.799,-73.097,-178.395,10.015,149.558
C01460=1109.832,256.551,-73.069,-178.397,10.012,149.558
C01461=1109.836,256.302,-73.039,-178.400,10.010,149.558
C01462=1109.840,256.053,-73.011,-178.403,10.007,149.558
C01463=1109.844,255.842,-72.986,-178.405,10.005,149.558
C01464=1109.848,255.629,-72.961,-178.407,10.002,149.558
C01465=1109.851,255.416,-72.936,-178.409,10.000,149.558
C01466=1109.855,255.203,-72.912,-178.410,9.999,149.558
C01467=1109.858,254.991,-72.887,-178.413,9.997,149.558
C01468=1109.862,254.778,-72.863,-178.415,9.995,149.558
C01469=1109.866,254.566,-72.838,-178.417,9.992,149.558
C01470=1109.869,254.352,-72.813,-178.419,9.990,149.558
C01471=1109.873,254.105,-72.785,-178.422,9.988,149.558
C01472=1109.878,253.856,-72.756,-178.424,9.986,149.558
C01473=1109.882,253.607,-72.727,-178.427,9.984,149.558
C01474=1109.886,253.360,-72.699,-178.430,9.981,149.559
C01475=1109.891,253.111,-72.670,-178.432,9.979,149.559
C01476=1109.894,252.863,-72.641,-178.435,9.976,149.559
C01477=1109.899,252.615,-72.613,-178.438,9.973,149.559
C01478=1109.904,252.366,-72.584,-178.440,9.971,149.559
C01479=1109.907,252.118,-72.555,-178.444,9.969,149.559
C01480=1109.912,251.870,-72.527,-178.446,9.966,149.559
C01481=1109.916,251.621,-72.499,-178.449,9.964,149.560
C01482=1109.920,251.373,-72.469,-178.452,9.962,149.560
C01483=1109.924,251.124,-72.441,-178.455,9.959,149.560
C01484=1109.929,250.876,-72.413,-178.458,9.956,149.560
C01485=1109.933,250.628,-72.384,-178.461,9.954,149.560
C01486=1109.938,250.380,-72.355,-178.464,9.951,149.561
C01487=1109.942,250.131,-72.327,-178.467,9.949,149.561
C01488=1109.946,249.883,-72.298,-178.470,9.946,149.561
C01489=1109.950,249.635,-72.271,-178.473,9.943,149.561
C01490=1109.954,249.386,-72.241,-178.477,9.941,149.561
C01491=1109.958,249.138,-72.213,-178.480,9.937,149.561
C01492=1109.963,248.890,-72.185,-178.483,9.934,149.561
C01493=1109.967,248.641,-72.157,-178.486,9.932,149.561
C01494=1109.972,248.393,-72.128,-178.490,9.928,149.562
C01495=1109.976,248.144,-72.100,-178.493,9.925,149.562
C01496=1109.980,247.895,-72.071,-178.496,9.922,149.562
C01497=1109.985,247.648,-72.044,-178.499,9.919,149.562
C01498=1109.989,247.399,-72.014,-178.502,9.916,149.562
C01499=1109.993,247.151,-71.986,-178.504,9.913,149.562
C01500=1109.997,246.903,-71.958,-178.507,9.910,149.562
C01501=1110.002,246.655,-71.930,-178.508,9.907,149.562
C01502=1110.006,246.406,-71.902,-178.511,9.905,149.562
C01503=1110.010,246.158,-71.874,-178.514,9.901,149.562
C01504=1110.015,245.909,-71.845,-178.516,9.899,149.562
C01505=1110.018,245.661,-71.817,-178.519,9.896,149.562
C01506=1110.023,245.413,-71.789,-178.521,9.894,149.562
C01507=1110.027,245.164,-71.761,-178.523,9.891,149.562
C01508=1110.032,244.916,-71.733,-178.526,9.888,149.562
C01509=1110.036,244.667,-71.705,-178.528,9.886,149.562
C01510=1110.041,244.419,-71.677,-178.531,9.883,149.562
C01511=1110.044,244.170,-71.649,-178.534,9.880,149.562
C01512=1110.049,243.922,-71.621,-178.535,9.878,149.562
C01513=1110.053,243.673,-71.592,-178.538,9.875,149.562
C01514=1110.058,243.426,-71.564,-178.540,9.873,149.562
C01515=1110.061,243.177,-71.536,-178.543,9.870,149.562
C01516=1110.066,242.929,-71.509,-178.546,9.867,149.562
C01517=1110.070,242.680,-71.480,-178.548,9.865,149.562
C01518=1110.075,242.432,-71.453,-178.551,9.862,149.562
C01519=1110.078,242.219,-71.429,-178.553,9.860,149.562
C01520=1110.082,242.006,-71.405,-178.555,9.858,149.562
C01521=1110.086,241.794,-71.381,-178.557,9.855,149.562
C01522=1110.090,241.581,-71.357,-178.559,9.853,149.562
C01523=1110.093,241.368,-71.333,-178.561,9.851,149.562
C01524=1110.097,241.155,-71.309,-178.564,9.848,149.562
C01525=1110.101,240.943,-71.285,-178.566,9.846,149.562
C01526=1110.104,240.730,-71.261,-178.568,9.844,149.562
C01527=1110.108,240.481,-71.233,-178.571,9.842,149.562
C01528=1110.113,240.233,-71.206,-178.573,9.839,149.562
C01529=1110.118,239.984,-71.178,-178.576,9.836,149.562
C01530=1110.122,239.736,-71.150,-178.579,9.834,149.563
C01531=1110.126,239.487,-71.123,-178.581,9.831,149.563
C01532=1110.130,239.239,-71.094,-178.584,9.828,149.563
C01533=1110.134,238.991,-71.067,-178.586,9.826,149.563
C01534=1110.139,238.742,-71.040,-178.589,9.824,149.563
C01535=1110.143,238.494,-71.011,-178.592,9.821,149.563
C01536=1110.148,238.246,-70.983,-178.594,9.818,149.563
C01537=1110.152,237.996,-70.956,-178.597,9.816,149.563
C01538=1110.156,237.749,-70.928,-178.600,9.813,149.563
C01539=1110.161,237.500,-70.901,-178.602,9.811,149.563
C01540=1110.165,237.252,-70.873,-178.605,9.808,149.563
C01541=1110.169,237.004,-70.845,-178.608,9.805,149.563
C01542=1110.174,236.755,-70.818,-178.610,9.803,149.563
C01543=1110.177,236.507,-70.790,-178.613,9.800,149.564
C01544=1110.182,236.258,-70.763,-178.616,9.798,149.564
C01545=1110.186,236.010,-70.735,-178.618,9.795,149.564
C01546=1110.190,235.761,-70.707,-178.621,9.793,149.564
C01547=1110.195,235.513,-70.680,-178.624,9.790,149.564
C01548=1110.199,235.265,-70.653,-178.627,9.787,149.564
C01549=1110.203,235.016,-70.624,-178.630,9.784,149.564
C01550=1110.208,234.768,-70.597,-178.632,9.782,149.564
C01551=1110.212,234.519,-70.570,-178.634,9.779,149.564
C01552=1110.216,234.270,-70.542,-178.637,9.776,149.564
C01553=1110.221,234.022,-70.515,-178.640,9.774,149.564
C01554=1110.225,233.774,-70.487,-178.642,9.771,149.564
C01555=1110.229,233.525,-70.460,-178.645,9.769,149.565
C01556=1110.234,233.276,-70.433,-178.648,9.766,149.565
C01557=1110.238,233.029,-70.405,-178.651,9.763,149.565
C01558=1110.243,232.780,-70.378,-178.654,9.760,149.565
C01559=1110.247,232.531,-70.351,-178.656,9.758,149.565
C01560=1110.251,232.283,-70.323,-178.659,9.755,149.565
C01561=1110.256,232.034,-70.296,-178.661,9.752,149.565
C01562=1110.260,231.785,-70.268,-178.664,9.749,149.565
C01563=1110.264,231.537,-70.242,-178.667,9.747,149.565
C01564=1110.268,231.289,-70.214,-178.670,9.744,149.565
C01565=1110.273,231.041,-70.187,-178.673,9.741,149.565
C01566=1110.277,230.792,-70.160,-178.675,9.738,149.565
C01567=1110.282,230.543,-70.132,-178.678,9.735,149.565
C01568=1110.286,230.295,-70.105,-178.681,9.732,149.565
C01569=1110.291,230.047,-70.078,-178.683,9.730,149.565
C01570=1110.295,229.798,-70.051,-178.686,9.727,149.565
C01571=1110.299,229.549,-70.024,-178.689,9.724,149.565
C01572=1110.303,229.301,-69.997,-178.692,9.721,149.565
C01573=1110.308,229.052,-69.970,-178.694,9.718,149.565
C01574=1110.312,228.804,-69.942,-178.697,9.715,149.566
C01575=1110.316,228.591,-69.920,-178.700,9.712,149.565
C01576=1110.319,228.378,-69.896,-178.701,9.710,149.565
C01577=1110.323,228.165,-69.873,-178.704,9.707,149.566
C01578=1110.327,227.953,-69.849,-178.706,9.705,149.565
C01579=1110.330,227.740,-69.827,-178.708,9.703,149.565
C01580=1110.334,227.527,-69.803,-178.711,9.699,149.565
C01581=1110.338,227.313,-69.780,-178.713,9.698,149.566
C01582=1110.343,227.101,-69.757,-178.716,9.694,149.565
C01583=1110.346,226.852,-69.730,-178.718,9.691,149.565
C01584=1110.351,226.604,-69.703,-178.720,9.689,149.565
C01585=1110.355,226.355,-69.676,-178.722,9.686,149.565
C01586=1110.360,226.107,-69.649,-178.725,9.683,149.565
C01587=1110.364,225.859,-69.623,-178.728,9.680,149.565
C01588=1110.368,225.610,-69.596,-178.730,9.677,149.565
C01589=1110.373,225.362,-69.569,-178.733,9.674,149.565
C01590=1110.376,225.113,-69.542,-178.735,9.671,149.565
C01591=1110.381,224.864,-69.515,-178.738,9.668,149.565
C01592=1110.386,224.616,-69.488,-178.741,9.664,149.565
C01593=1110.390,224.367,-69.461,-178.743,9.661,149.565
C01594=1110.395,224.118,-69.435,-178.746,9.658,149.565
C01595=1110.399,223.870,-69.408,-178.748,9.655,149.565
C01596=1110.403,223.622,-69.381,-178.751,9.652,149.565
C01597=1110.408,223.373,-69.354,-178.753,9.649,149.565
C01598=1110.412,223.125,-69.328,-178.756,9.646,149.565
C01599=1110.416,222.876,-69.301,-178.758,9.643,149.564
C01600=1110.421,222.628,-69.275,-178.760,9.640,149.564
C01601=1110.425,222.379,-69.248,-178.763,9.637,149.564
C01602=1110.430,222.131,-69.221,-178.765,9.634,149.564
C01603=1110.434,221.883,-69.194,-178.768,9.631,149.564
C01604=1110.438,221.633,-69.168,-178.770,9.628,149.564
C01605=1110.442,221.384,-69.141,-178.773,9.625,149.564
C01606=1110.447,221.136,-69.114,-178.775,9.621,149.564
C01607=1110.451,220.888,-69.088,-178.777,9.618,149.564
C01608=1110.456,220.639,-69.061,-178.780,9.615,149.564
C01609=1110.460,220.391,-69.035,-178.782,9.613,149.564
C01610=1110.464,220.142,-69.008,-178.784,9.610,149.564
C01611=1110.468,219.893,-68.982,-178.787,9.607,149.564
C01612=1110.473,219.645,-68.955,-178.789,9.603,149.563
C01613=1110.477,219.397,-68.928,-178.791,9.600,149.563
C01614=1110.482,219.147,-68.902,-178.794,9.597,149.563
C01615=1110.486,218.899,-68.876,-178.797,9.594,149.563
C01616=1110.491,218.650,-68.849,-178.798,9.591,149.563
C01617=1110.495,218.402,-68.823,-178.801,9.588,149.563
C01618=1110.499,218.154,-68.796,-178.803,9.585,149.563
C01619=1110.504,217.905,-68.770,-178.806,9.582,149.563
C01620=1110.508,217.657,-68.744,-178.808,9.579,149.563
C01621=1110.513,217.408,-68.718,-178.810,9.576,149.562
C01622=1110.517,217.160,-68.691,-178.812,9.573,149.562
C01623=1110.521,216.911,-68.665,-178.815,9.570,149.562
C01624=1110.526,216.663,-68.638,-178.817,9.567,149.562
C01625=1110.530,216.414,-68.613,-178.819,9.564,149.562
C01626=1110.535,216.165,-68.585,-178.821,9.561,149.562
C01627=1110.539,215.916,-68.560,-178.824,9.558,149.562
C01628=1110.543,215.668,-68.533,-178.826,9.555,149.562
C01629=1110.548,215.419,-68.507,-178.828,9.552,149.562
C01630=1110.552,215.171,-68.480,-178.830,9.549,149.561
C01631=1110.556,214.958,-68.459,-178.832,9.546,149.561
C01632=1110.560,214.745,-68.436,-178.834,9.544,149.561
C01633=1110.563,214.531,-68.414,-178.836,9.542,149.561
C01634=1110.568,214.318,-68.391,-178.838,9.539,149.561
C01635=1110.571,214.106,-68.368,-178.840,9.536,149.561
C01636=1110.575,213.893,-68.346,-178.842,9.534,149.561
C01637=1110.579,213.679,-68.324,-178.844,9.531,149.561
C01638=1110.582,213.466,-68.301,-178.846,9.529,149.561
C01639=1110.587,213.219,-68.275,-178.849,9.525,149.561
C01640=1110.591,212.970,-68.249,-178.852,9.522,149.561
C01641=1110.596,212.721,-68.223,-178.854,9.519,149.561
C01642=1110.600,212.472,-68.198,-178.858,9.516,149.561
C01643=1110.604,212.224,-68.171,-178.860,9.513,149.561
C01644=1110.609,211.975,-68.145,-178.863,9.509,149.561
C01645=1110.614,211.727,-68.119,-178.866,9.506,149.561
C01646=1110.618,211.478,-68.094,-178.869,9.503,149.561
C01647=1110.622,211.230,-68.067,-178.872,9.500,149.561
C01648=1110.626,210.981,-68.041,-178.875,9.497,149.561
C01649=1110.631,210.732,-68.015,-178.878,9.493,149.561
C01650=1110.635,210.483,-67.989,-178.881,9.491,149.561
C01651=1110.640,210.235,-67.964,-178.883,9.488,149.561
C01652=1110.644,209.986,-67.938,-178.887,9.484,149.561
C01653=1110.648,209.738,-67.912,-178.890,9.481,149.561
C01654=1110.652,209.489,-67.886,-178.892,9.478,149.561
C01655=1110.657,209.241,-67.861,-178.895,9.475,149.561
C01656=1110.662,208.992,-67.834,-178.898,9.473,149.562
C01657=1110.666,208.743,-67.808,-178.902,9.469,149.561
C01658=1110.671,208.494,-67.783,-178.904,9.466,149.562
C01659=1110.675,208.246,-67.757,-178.907,9.463,149.562
C01660=1110.680,207.997,-67.732,-178.910,9.461,149.562
C01661=1110.684,207.748,-67.706,-178.913,9.457,149.562
C01662=1110.688,207.500,-67.680,-178.916,9.455,149.562
C01663=1110.693,207.251,-67.655,-178.919,9.452,149.562
C01664=1110.697,207.003,-67.629,-178.922,9.448,149.562
C01665=1110.701,206.754,-67.603,-178.925,9.445,149.562
C01666=1110.706,206.505,-67.577,-178.928,9.443,149.562
C01667=1110.710,206.257,-67.552,-178.931,9.440,149.562
C01668=1110.715,206.008,-67.526,-178.933,9.437,149.562
C01669=1110.719,205.759,-67.501,-178.936,9.434,149.563
C01670=1110.724,205.511,-67.475,-178.939,9.431,149.563
C01671=1110.728,205.262,-67.450,-178.942,9.428,149.563
C01672=1110.732,205.013,-67.424,-178.945,9.425,149.563
C01673=1110.737,204.765,-67.399,-178.948,9.423,149.563
C01674=1110.742,204.516,-67.373,-178.951,9.420,149.563
C01675=1110.746,204.267,-67.347,-178.954,9.417,149.563
C01676=1110.751,204.019,-67.322,-178.956,9.414,149.563
C01677=1110.755,203.770,-67.297,-178.959,9.411,149.563
C01678=1110.759,203.521,-67.271,-178.962,9.409,149.563
C01679=1110.764,203.273,-67.246,-178.964,9.405,149.563
C01680=1110.768,203.024,-67.220,-178.967,9.403,149.564
C01681=1110.774,202.775,-67.195,-178.971,9.399,149.564
C01682=1110.778,202.527,-67.170,-178.974,9.396,149.564
C01683=1110.782,202.278,-67.144,-178.976,9.393,149.564
C01684=1110.786,202.030,-67.119,-178.979,9.391,149.564
C01685=1110.791,201.780,-67.094,-178.982,9.387,149.564
C01686=1110.795,201.532,-67.069,-178.985,9.385,149.564
C01687=1110.799,201.318,-67.047,-178.987,9.382,149.564
C01688=1110.803,201.106,-67.025,-178.989,9.380,149.564
C01689=1110.806,200.892,-67.003,-178.992,9.377,149.564
C01690=1110.810,200.679,-66.982,-178.994,9.375,149.564
C01691=1110.814,200.467,-66.960,-178.996,9.372,149.564
C01692=1110.818,200.253,-66.939,-178.999,9.370,149.564
C01693=1110.822,200.040,-66.917,-179.001,9.367,149.564
C01694=1110.826,199.827,-66.896,-179.003,9.365,149.564
C01695=1110.830,199.578,-66.870,-179.006,9.362,149.564
C01696=1110.835,199.330,-66.846,-179.009,9.359,149.564
C01697=1110.839,199.081,-66.820,-179.012,9.356,149.564
C01698=1110.844,198.832,-66.796,-179.014,9.353,149.564
C01699=1110.848,198.583,-66.770,-179.017,9.350,149.564
C01700=1110.852,198.334,-66.745,-179.020,9.347,149.564
C01701=1110.857,198.086,-66.720,-179.022,9.344,149.564
C01702=1110.861,197.837,-66.695,-179.025,9.341,149.564
C01703=1110.866,197.588,-66.670,-179.027,9.338,149.564
C01704=1110.870,197.339,-66.645,-179.030,9.335,149.564
C01705=1110.875,197.091,-66.620,-179.033,9.332,149.564
C01706=1110.879,196.842,-66.595,-179.035,9.329,149.564
C01707=1110.884,196.593,-66.571,-179.038,9.326,149.564
C01708=1110.888,196.345,-66.545,-179.040,9.323,149.564
C01709=1110.893,196.096,-66.520,-179.042,9.319,149.564
C01710=1110.897,195.847,-66.495,-179.044,9.317,149.564
C01711=1110.902,195.599,-66.471,-179.047,9.314,149.564
C01712=1110.906,195.350,-66.446,-179.048,9.311,149.564
C01713=1110.910,195.101,-66.421,-179.051,9.308,149.564
C01714=1110.916,194.853,-66.396,-179.053,9.306,149.564
C01715=1110.919,194.604,-66.372,-179.055,9.303,149.564
C01716=1110.924,194.356,-66.346,-179.057,9.300,149.563
C01717=1110.929,194.106,-66.321,-179.059,9.297,149.563
C01718=1110.933,193.858,-66.297,-179.061,9.294,149.563
C01719=1110.938,193.608,-66.272,-179.064,9.291,149.563
C01720=1110.942,193.360,-66.247,-179.065,9.289,149.563
C01721=1110.947,193.112,-66.223,-179.068,9.286,149.563
C01722=1110.951,192.863,-66.198,-179.069,9.283,149.563
C01723=1110.956,192.614,-66.173,-179.072,9.280,149.563
C01724=1110.960,192.365,-66.148,-179.074,9.278,149.563
C01725=1110.964,192.117,-66.124,-179.076,9.275,149.563
C01726=1110.969,191.868,-66.099,-179.079,9.272,149.563
C01727=1110.973,191.619,-66.075,-179.081,9.269,149.563
C01728=1110.978,191.370,-66.050,-179.083,9.266,149.563
C01729=1110.982,191.121,-66.025,-179.085,9.264,149.562
C01730=1110.987,190.873,-66.000,-179.088,9.261,149.562
C01731=1110.991,190.625,-65.976,-179.090,9.258,149.562
C01732=1110.996,190.375,-65.951,-179.092,9.255,149.562
C01733=1111.000,190.127,-65.927,-179.095,9.252,149.562
C01734=1111.005,189.878,-65.902,-179.097,9.250,149.562
C01735=1111.009,189.629,-65.878,-179.099,9.247,149.562
C01736=1111.014,189.380,-65.853,-179.101,9.244,149.562
C01737=1111.019,189.132,-65.829,-179.104,9.241,149.562
C01738=1111.023,188.882,-65.804,-179.106,9.238,149.562
C01739=1111.028,188.634,-65.780,-179.108,9.236,149.562
C01740=1111.032,188.385,-65.756,-179.110,9.233,149.562
C01741=1111.037,188.136,-65.731,-179.112,9.230,149.562
C01742=1111.041,187.888,-65.707,-179.115,9.227,149.562
C01743=1111.045,187.674,-65.686,-179.117,9.225,149.562
C01744=1111.049,187.461,-65.664,-179.119,9.223,149.562
C01745=1111.053,187.248,-65.644,-179.121,9.220,149.562
C01746=1111.057,187.034,-65.622,-179.122,9.218,149.562
C01747=1111.060,186.821,-65.602,-179.125,9.215,149.562
C01748=1111.064,186.608,-65.581,-179.127,9.212,149.562
C01749=1111.068,186.395,-65.560,-179.129,9.210,149.562
C01750=1111.072,186.182,-65.539,-179.131,9.208,149.562
C01751=1111.077,185.933,-65.515,-179.133,9.205,149.562
C01752=1111.081,185.684,-65.490,-179.135,9.202,149.562
C01753=1111.085,185.436,-65.466,-179.138,9.199,149.561
C01754=1111.091,185.186,-65.442,-179.140,9.196,149.561
C01755=1111.095,184.938,-65.418,-179.143,9.193,149.561
C01756=1111.099,184.689,-65.394,-179.145,9.191,149.561
C01757=1111.104,184.440,-65.369,-179.147,9.188,149.561
C01758=1111.108,184.192,-65.345,-179.150,9.184,149.561
C01759=1111.113,183.943,-65.321,-179.151,9.182,149.561
C01760=1111.117,183.693,-65.297,-179.154,9.179,149.561
C01761=1111.122,183.445,-65.272,-179.157,9.176,149.561
C01762=1111.126,183.196,-65.248,-179.159,9.173,149.561
C01763=1111.131,182.948,-65.224,-179.161,9.170,149.561
C01764=1111.135,182.699,-65.201,-179.163,9.167,149.561
C01765=1111.140,182.449,-65.176,-179.166,9.164,149.561
C01766=1111.144,182.201,-65.152,-179.169,9.161,149.561
C01767=1111.149,181.953,-65.128,-179.171,9.158,149.561
C01768=1111.153,181.704,-65.104,-179.174,9.155,149.561
C01769=1111.158,181.455,-65.080,-179.175,9.153,149.561
C01770=1111.162,181.206,-65.055,-179.178,9.150,149.561
C01771=1111.167,180.957,-65.032,-179.180,9.146,149.561
C01772=1111.171,180.708,-65.008,-179.183,9.143,149.561
C01773=1111.176,180.460,-64.984,-179.186,9.140,149.561
C01774=1111.181,180.211,-64.960,-179.188,9.137,149.561
C01775=1111.184,179.962,-64.936,-179.190,9.134,149.560
C01776=1111.190,179.712,-64.912,-179.192,9.131,149.560
C01777=1111.194,179.464,-64.888,-179.195,9.128,149.560
C01778=1111.199,179.216,-64.864,-179.197,9.125,149.560
C01779=1111.203,178.967,-64.840,-179.200,9.122,149.560
C01780=1111.208,178.718,-64.816,-179.201,9.119,149.560
C01781=1111.212,178.469,-64.793,-179.204,9.116,149.560
C01782=1111.216,178.220,-64.769,-179.206,9.113,149.560
C01783=1111.221,177.971,-64.745,-179.208,9.110,149.560
C01784=1111.225,177.723,-64.721,-179.210,9.107,149.560
C01785=1111.230,177.474,-64.698,-179.213,9.104,149.560
C01786=1111.234,177.225,-64.674,-179.214,9.101,149.559
C01787=1111.239,176.976,-64.650,-179.217,9.098,149.559
C01788=1111.244,176.727,-64.626,-179.219,9.095,149.559
C01789=1111.249,176.478,-64.602,-179.221,9.092,149.559
C01790=1111.253,176.230,-64.578,-179.223,9.089,149.559
C01791=1111.258,175.981,-64.555,-179.226,9.086,149.559
C01792=1111.263,175.732,-64.532,-179.227,9.084,149.559
C01793=1111.266,175.483,-64.507,-179.230,9.080,149.559
C01794=1111.271,175.234,-64.484,-179.232,9.077,149.559
C01795=1111.276,174.985,-64.460,-179.234,9.075,149.558
C01796=1111.280,174.736,-64.436,-179.236,9.071,149.558
C01797=1111.285,174.487,-64.413,-179.239,9.068,149.558
C01798=1111.289,174.239,-64.389,-179.240,9.066,149.558
C01799=1111.293,174.025,-64.369,-179.242,9.063,149.558
C01800=1111.297,173.812,-64.349,-179.244,9.061,149.558
